Yaskawa INFORM job: DEMO_ROOF_UPPER_0625_3PAINT_58.JBI

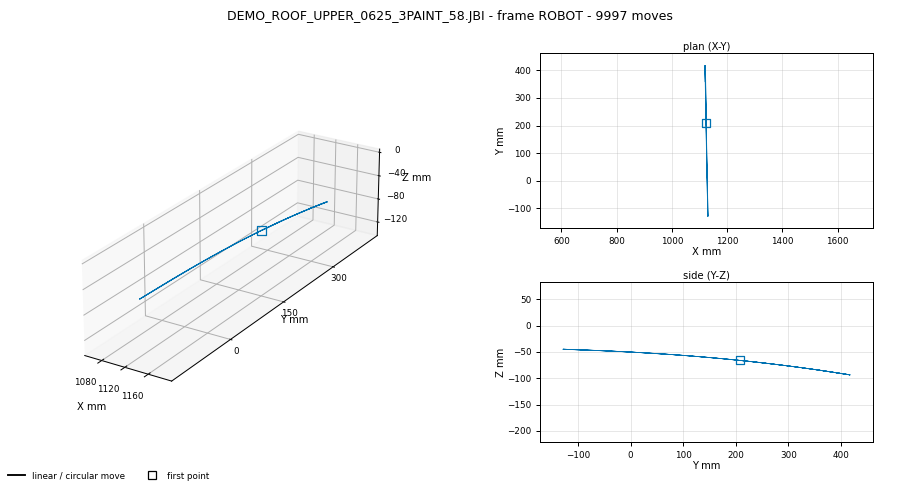
[picture p0: tool path of DEMO_ROOF_UPPER_0625_3PAINT_58.JBI in frame ROBOT, 9997 of 9997 moves have a stored position in this frame; points joined in program order, loops and branches not executed]
/JOB
//NAME DEMO_ROOF_UPPER_0625_3PAINT58
//POS
///NPOS 9997,0,0,0,0,0
///TOOL 0
///USER 0
///POSTYPE ROBOT
///RECTAN
///RCONF 1,0,0,0,0,0,0,0,0,0,0,0,0,0,0,0,0,0,0,0,0,0,0,0
C00000=1124.539,208.417,-65.917,-178.958,9.435,149.569
C00001=1124.534,208.666,-65.943,-178.955,9.438,149.569
C00002=1124.530,208.915,-65.969,-178.953,9.440,149.568
C00003=1124.525,209.163,-65.994,-178.950,9.443,149.569
C00004=1124.521,209.412,-66.020,-178.948,9.447,149.569
C00005=1124.516,209.661,-66.045,-178.945,9.449,149.568
C00006=1124.512,209.910,-66.070,-178.943,9.452,149.569
C00007=1124.507,210.158,-66.096,-178.941,9.454,149.569
C00008=1124.503,210.407,-66.122,-178.938,9.457,149.569
C00009=1124.498,210.655,-66.147,-178.937,9.459,149.569
C00010=1124.493,210.904,-66.174,-178.934,9.462,149.569
C00011=1124.489,211.153,-66.199,-178.932,9.465,149.569
C00012=1124.484,211.401,-66.225,-178.930,9.468,149.569
C00013=1124.480,211.650,-66.250,-178.928,9.470,149.569
C00014=1124.477,211.864,-66.272,-178.926,9.473,149.569
C00015=1124.472,212.078,-66.295,-178.924,9.475,149.569
C00016=1124.469,212.292,-66.316,-178.922,9.477,149.569
C00017=1124.465,212.505,-66.339,-178.920,9.480,149.569
C00018=1124.461,212.719,-66.360,-178.919,9.482,149.569
C00019=1124.457,212.933,-66.383,-178.917,9.485,149.569
C00020=1124.454,213.147,-66.405,-178.915,9.487,149.569
C00021=1124.450,213.361,-66.428,-178.914,9.489,149.570
C00022=1124.445,213.609,-66.453,-178.912,9.492,149.570
C00023=1124.441,213.858,-66.479,-178.910,9.494,149.570
C00024=1124.437,214.107,-66.505,-178.908,9.497,149.570
C00025=1124.433,214.356,-66.531,-178.906,9.500,149.570
C00026=1124.428,214.604,-66.556,-178.904,9.503,149.570
C00027=1124.423,214.853,-66.582,-178.902,9.505,149.570
C00028=1124.419,215.102,-66.608,-178.900,9.509,149.571
C00029=1124.414,215.351,-66.634,-178.898,9.511,149.571
C00030=1124.410,215.598,-66.660,-178.896,9.514,149.571
C00031=1124.406,215.847,-66.686,-178.894,9.517,149.571
C00032=1124.401,216.096,-66.711,-178.892,9.520,149.571
C00033=1124.396,216.345,-66.738,-178.890,9.522,149.571
C00034=1124.392,216.594,-66.763,-178.888,9.526,149.571
C00035=1124.387,216.842,-66.789,-178.885,9.529,149.571
C00036=1124.383,217.090,-66.815,-178.883,9.531,149.571
C00037=1124.379,217.339,-66.841,-178.881,9.535,149.572
C00038=1124.374,217.588,-66.867,-178.879,9.538,149.572
C00039=1124.370,217.837,-66.893,-178.877,9.540,149.572
C00040=1124.366,218.085,-66.920,-178.874,9.543,149.572
C00041=1124.361,218.333,-66.945,-178.872,9.547,149.572
C00042=1124.356,218.582,-66.971,-178.870,9.550,149.572
C00043=1124.352,218.830,-66.998,-178.868,9.552,149.572
C00044=1124.348,219.079,-67.024,-178.865,9.555,149.572
C00045=1124.344,219.328,-67.049,-178.863,9.559,149.573
C00046=1124.339,219.576,-67.076,-178.861,9.562,149.573
C00047=1124.335,219.825,-67.102,-178.858,9.565,149.573
C00048=1124.330,220.073,-67.128,-178.856,9.568,149.573
C00049=1124.326,220.322,-67.155,-178.853,9.571,149.573
C00050=1124.321,220.570,-67.180,-178.850,9.574,149.573
C00051=1124.317,220.819,-67.206,-178.848,9.577,149.573
C00052=1124.313,221.068,-67.233,-178.845,9.580,149.573
C00053=1124.308,221.317,-67.259,-178.843,9.584,149.573
C00054=1124.304,221.565,-67.285,-178.840,9.587,149.573
C00055=1124.299,221.814,-67.312,-178.838,9.590,149.573
C00056=1124.296,222.062,-67.338,-178.835,9.593,149.573
C00057=1124.291,222.311,-67.365,-178.832,9.597,149.573
C00058=1124.286,222.559,-67.391,-178.830,9.600,149.573
C00059=1124.282,222.807,-67.416,-178.827,9.603,149.573
C00060=1124.277,223.056,-67.443,-178.825,9.606,149.573
C00061=1124.273,223.305,-67.469,-178.822,9.609,149.573
C00062=1124.268,223.553,-67.496,-178.818,9.613,149.573
C00063=1124.264,223.802,-67.522,-178.816,9.616,149.574
C00064=1124.259,224.051,-67.549,-178.813,9.619,149.574
C00065=1124.255,224.299,-67.575,-178.810,9.623,149.574
C00066=1124.251,224.548,-67.602,-178.807,9.626,149.574
C00067=1124.247,224.796,-67.628,-178.805,9.629,149.574
C00068=1124.242,225.045,-67.655,-178.801,9.632,149.573
C00069=1124.238,225.293,-67.681,-178.799,9.635,149.574
C00070=1124.234,225.507,-67.704,-178.796,9.638,149.574
C00071=1124.230,225.721,-67.727,-178.793,9.641,149.573
C00072=1124.226,225.935,-67.750,-178.791,9.644,149.574
C00073=1124.222,226.149,-67.773,-178.788,9.647,149.573
C00074=1124.219,226.362,-67.795,-178.786,9.649,149.573
C00075=1124.215,226.576,-67.818,-178.783,9.652,149.573
C00076=1124.212,226.789,-67.842,-178.780,9.655,149.573
C00077=1124.208,227.003,-67.864,-178.777,9.658,149.573
C00078=1124.203,227.252,-67.891,-178.774,9.662,149.573
C00079=1124.199,227.500,-67.917,-178.771,9.665,149.573
C00080=1124.194,227.749,-67.944,-178.768,9.668,149.573
C00081=1124.189,227.997,-67.971,-178.765,9.672,149.573
C00082=1124.186,228.246,-67.998,-178.762,9.675,149.573
C00083=1124.181,228.494,-68.025,-178.758,9.678,149.573
C00084=1124.177,228.743,-68.051,-178.754,9.682,149.573
C00085=1124.173,228.992,-68.078,-178.751,9.684,149.573
C00086=1124.168,229.241,-68.105,-178.748,9.688,149.573
C00087=1124.164,229.489,-68.131,-178.744,9.692,149.572
C00088=1124.159,229.737,-68.159,-178.741,9.695,149.572
C00089=1124.155,229.986,-68.186,-178.738,9.698,149.572
C00090=1124.150,230.234,-68.213,-178.734,9.701,149.572
C00091=1124.146,230.482,-68.239,-178.731,9.705,149.572
C00092=1124.141,230.731,-68.266,-178.727,9.708,149.572
C00093=1124.137,230.979,-68.293,-178.724,9.711,149.572
C00094=1124.133,231.228,-68.320,-178.721,9.715,149.572
C00095=1124.129,231.477,-68.347,-178.718,9.717,149.572
C00096=1124.124,231.725,-68.374,-178.714,9.721,149.571
C00097=1124.120,231.974,-68.401,-178.711,9.723,149.571
C00098=1124.115,232.222,-68.428,-178.707,9.727,149.571
C00099=1124.111,232.470,-68.455,-178.704,9.730,149.571
C00100=1124.107,232.720,-68.482,-178.701,9.732,149.571
C00101=1124.103,232.967,-68.510,-178.698,9.736,149.571
C00102=1124.098,233.216,-68.537,-178.695,9.739,149.570
C00103=1124.093,233.464,-68.564,-178.692,9.741,149.570
C00104=1124.089,233.713,-68.591,-178.689,9.744,149.570
C00105=1124.085,233.962,-68.618,-178.686,9.747,149.570
C00106=1124.081,234.210,-68.645,-178.682,9.750,149.570
C00107=1124.076,234.458,-68.673,-178.679,9.753,149.570
C00108=1124.072,234.707,-68.700,-178.676,9.756,149.570
C00109=1124.068,234.956,-68.727,-178.673,9.759,149.570
C00110=1124.063,235.204,-68.754,-178.670,9.761,149.569
C00111=1124.059,235.452,-68.782,-178.668,9.764,149.570
C00112=1124.054,235.701,-68.809,-178.665,9.767,149.569
C00113=1124.051,235.950,-68.836,-178.662,9.770,149.569
C00114=1124.046,236.198,-68.864,-178.660,9.772,149.569
C00115=1124.042,236.446,-68.891,-178.657,9.775,149.569
C00116=1124.037,236.695,-68.918,-178.654,9.777,149.569
C00117=1124.033,236.943,-68.946,-178.651,9.780,149.569
C00118=1124.028,237.192,-68.973,-178.648,9.783,149.569
C00119=1124.024,237.440,-69.000,-178.646,9.785,149.569
C00120=1124.019,237.688,-69.028,-178.643,9.788,149.569
C00121=1124.015,237.937,-69.055,-178.640,9.791,149.568
C00122=1124.011,238.185,-69.083,-178.638,9.793,149.568
C00123=1124.006,238.434,-69.110,-178.635,9.796,149.568
C00124=1124.003,238.682,-69.138,-178.632,9.799,149.568
C00125=1123.998,238.931,-69.165,-178.630,9.801,149.568
C00126=1123.994,239.145,-69.190,-178.628,9.803,149.568
C00127=1123.990,239.358,-69.213,-178.626,9.805,149.568
C00128=1123.986,239.571,-69.236,-178.624,9.807,149.568
C00129=1123.983,239.785,-69.260,-178.622,9.809,149.568
C00130=1123.979,239.998,-69.284,-178.620,9.811,149.568
C00131=1123.976,240.212,-69.308,-178.617,9.813,149.568
C00132=1123.972,240.426,-69.331,-178.616,9.816,149.568
C00133=1123.968,240.640,-69.355,-178.613,9.818,149.568
C00134=1123.963,240.888,-69.383,-178.611,9.820,149.568
C00135=1123.959,241.137,-69.411,-178.609,9.822,149.568
C00136=1123.955,241.385,-69.438,-178.606,9.825,149.568
C00137=1123.951,241.633,-69.466,-178.604,9.827,149.568
C00138=1123.947,241.882,-69.494,-178.602,9.829,149.568
C00139=1123.942,242.130,-69.521,-178.600,9.832,149.568
C00140=1123.937,242.379,-69.549,-178.597,9.835,149.568
C00141=1123.933,242.627,-69.577,-178.596,9.837,149.568
C00142=1123.929,242.875,-69.605,-178.594,9.839,149.568
C00143=1123.925,243.124,-69.632,-178.592,9.842,149.568
C00144=1123.920,243.372,-69.660,-178.590,9.844,149.568
C00145=1123.917,243.621,-69.688,-178.588,9.846,149.568
C00146=1123.912,243.869,-69.715,-178.586,9.848,149.568
C00147=1123.907,244.117,-69.744,-178.584,9.851,149.568
C00148=1123.903,244.366,-69.772,-178.582,9.853,149.568
C00149=1123.898,244.614,-69.799,-178.580,9.855,149.568
C00150=1123.895,244.863,-69.827,-178.578,9.858,149.568
C00151=1123.890,245.111,-69.855,-178.577,9.860,149.568
C00152=1123.886,245.360,-69.884,-178.575,9.863,149.568
C00153=1123.881,245.608,-69.911,-178.573,9.865,149.568
C00154=1123.877,245.856,-69.938,-178.572,9.866,149.568
C00155=1123.873,246.105,-69.967,-178.570,9.869,149.569
C00156=1123.869,246.353,-69.994,-178.568,9.871,149.569
C00157=1123.864,246.602,-70.022,-178.566,9.874,149.569
C00158=1123.860,246.850,-70.050,-178.565,9.876,149.569
C00159=1123.856,247.099,-70.078,-178.563,9.878,149.569
C00160=1123.851,247.346,-70.106,-178.562,9.881,149.569
C00161=1123.847,247.595,-70.135,-178.557,9.885,149.569
C00162=1123.842,247.844,-70.162,-178.552,9.889,149.569
C00163=1123.838,248.092,-70.190,-178.545,9.894,149.568
C00164=1123.833,248.341,-70.218,-178.540,9.899,149.568
C00165=1123.829,248.588,-70.246,-178.534,9.903,149.568
C00166=1123.825,248.837,-70.274,-178.529,9.908,149.567
C00167=1123.821,249.086,-70.303,-178.524,9.911,149.567
C00168=1123.817,249.334,-70.331,-178.519,9.915,149.566
C00169=1123.813,249.582,-70.359,-178.513,9.920,149.566
C00170=1123.808,249.831,-70.387,-178.509,9.923,149.566
C00171=1123.804,250.079,-70.415,-178.505,9.927,149.565
C00172=1123.799,250.327,-70.444,-178.500,9.931,149.565
C00173=1123.795,250.576,-70.472,-178.496,9.933,149.565
C00174=1123.790,250.824,-70.500,-178.492,9.937,149.564
C00175=1123.787,251.072,-70.529,-178.489,9.939,149.564
C00176=1123.783,251.321,-70.557,-178.485,9.943,149.564
C00177=1123.778,251.569,-70.586,-178.482,9.945,149.564
C00178=1123.774,251.817,-70.614,-178.478,9.948,149.563
C00179=1123.769,252.066,-70.642,-178.475,9.950,149.563
C00180=1123.765,252.313,-70.671,-178.472,9.953,149.563
C00181=1123.761,252.562,-70.700,-178.469,9.956,149.563
C00182=1123.756,252.776,-70.724,-178.467,9.958,149.563
C00183=1123.754,252.989,-70.748,-178.465,9.959,149.563
C00184=1123.750,253.203,-70.773,-178.463,9.961,149.563
C00185=1123.746,253.417,-70.797,-178.462,9.962,149.562
C00186=1123.742,253.629,-70.822,-178.460,9.965,149.563
C00187=1123.739,253.843,-70.846,-178.458,9.966,149.562
C00188=1123.735,254.057,-70.871,-178.457,9.967,149.562
C00189=1123.731,254.271,-70.896,-178.456,9.969,149.562
C00190=1123.727,254.518,-70.924,-178.455,9.970,149.563
C00191=1123.723,254.767,-70.953,-178.454,9.972,149.563
C00192=1123.719,255.016,-70.981,-178.453,9.973,149.563
C00193=1123.714,255.263,-71.010,-178.453,9.974,149.563
C00194=1123.710,255.512,-71.039,-178.453,9.975,149.563
C00195=1123.705,255.760,-71.067,-178.452,9.977,149.563
C00196=1123.701,256.008,-71.096,-178.451,9.978,149.564
C00197=1123.697,256.257,-71.124,-178.449,9.981,149.564
C00198=1123.692,256.505,-71.153,-178.446,9.984,149.563
C00199=1123.689,256.753,-71.182,-178.443,9.987,149.564
C00200=1123.684,257.002,-71.210,-178.440,9.990,149.563
C00201=1123.680,257.251,-71.239,-178.437,9.993,149.563
C00202=1123.676,257.498,-71.268,-178.434,9.995,149.563
C00203=1123.671,257.747,-71.296,-178.431,9.998,149.563
C00204=1123.667,257.995,-71.326,-178.428,10.001,149.563
C00205=1123.663,258.243,-71.353,-178.425,10.004,149.563
C00206=1123.658,258.492,-71.382,-178.422,10.006,149.563
C00207=1123.654,258.740,-71.412,-178.420,10.009,149.563
C00208=1123.650,258.988,-71.439,-178.416,10.013,149.563
C00209=1123.646,259.236,-71.469,-178.413,10.015,149.562
C00210=1123.641,259.485,-71.498,-178.410,10.018,149.562
C00211=1123.638,259.733,-71.526,-178.407,10.021,149.562
C00212=1123.633,259.981,-71.555,-178.404,10.024,149.562
C00213=1123.628,260.229,-71.584,-178.401,10.027,149.562
C00214=1123.624,260.478,-71.614,-178.398,10.030,149.562
C00215=1123.620,260.726,-71.642,-178.394,10.034,149.562
C00216=1123.616,260.975,-71.671,-178.391,10.036,149.562
C00217=1123.611,261.223,-71.700,-178.388,10.039,149.561
C00218=1123.607,261.471,-71.729,-178.384,10.042,149.561
C00219=1123.603,261.719,-71.759,-178.381,10.045,149.561
C00220=1123.599,261.968,-71.787,-178.377,10.048,149.561
C00221=1123.595,262.216,-71.816,-178.374,10.051,149.561
C00222=1123.590,262.464,-71.845,-178.370,10.054,149.561
C00223=1123.586,262.713,-71.874,-178.367,10.057,149.560
C00224=1123.581,262.961,-71.904,-178.363,10.060,149.560
C00225=1123.577,263.209,-71.933,-178.360,10.063,149.560
C00226=1123.574,263.457,-71.962,-178.357,10.066,149.560
C00227=1123.569,263.705,-71.990,-178.354,10.069,149.560
C00228=1123.565,263.954,-72.020,-178.350,10.072,149.559
C00229=1123.560,264.202,-72.049,-178.346,10.075,149.559
C00230=1123.556,264.450,-72.079,-178.343,10.078,149.559
C00231=1123.552,264.698,-72.108,-178.340,10.081,149.559
C00232=1123.548,264.947,-72.137,-178.337,10.083,149.559
C00233=1123.543,265.196,-72.166,-178.334,10.085,149.559
C00234=1123.539,265.443,-72.195,-178.332,10.087,149.559
C00235=1123.534,265.691,-72.225,-178.329,10.090,149.558
C00236=1123.530,265.940,-72.254,-178.327,10.092,149.558
C00237=1123.526,266.188,-72.284,-178.324,10.095,149.558
C00238=1123.522,266.401,-72.309,-178.322,10.097,149.558
C00239=1123.519,266.615,-72.334,-178.319,10.099,149.558
C00240=1123.515,266.828,-72.359,-178.317,10.101,149.558
C00241=1123.512,267.042,-72.384,-178.315,10.103,149.558
C00242=1123.508,267.255,-72.410,-178.313,10.105,149.558
C00243=1123.505,267.468,-72.435,-178.311,10.107,149.558
C00244=1123.501,267.682,-72.460,-178.308,10.109,149.558
C00245=1123.498,267.895,-72.486,-178.306,10.111,149.558
C00246=1123.494,268.143,-72.515,-178.303,10.114,149.558
C00247=1123.489,268.390,-72.544,-178.300,10.117,149.557
C00248=1123.485,268.639,-72.574,-178.298,10.119,149.557
C00249=1123.480,268.887,-72.604,-178.295,10.122,149.557
C00250=1123.476,269.136,-72.633,-178.292,10.124,149.557
C00251=1123.471,269.384,-72.663,-178.290,10.126,149.557
C00252=1123.467,269.632,-72.692,-178.287,10.129,149.557
C00253=1123.463,269.880,-72.722,-178.284,10.132,149.557
C00254=1123.459,270.129,-72.751,-178.281,10.135,149.557
C00255=1123.455,270.377,-72.781,-178.279,10.137,149.557
C00256=1123.450,270.625,-72.810,-178.276,10.139,149.556
C00257=1123.447,270.873,-72.840,-178.273,10.142,149.556
C00258=1123.442,271.121,-72.870,-178.270,10.145,149.556
C00259=1123.438,271.369,-72.899,-178.268,10.147,149.556
C00260=1123.433,271.618,-72.929,-178.265,10.150,149.556
C00261=1123.429,271.866,-72.959,-178.262,10.152,149.556
C00262=1123.425,272.114,-72.988,-178.259,10.155,149.556
C00263=1123.421,272.362,-73.018,-178.256,10.158,149.556
C00264=1123.417,272.610,-73.048,-178.253,10.160,149.555
C00265=1123.413,272.859,-73.077,-178.250,10.163,149.555
C00266=1123.408,273.107,-73.108,-178.247,10.166,149.555
C00267=1123.404,273.355,-73.137,-178.244,10.169,149.555
C00268=1123.400,273.603,-73.167,-178.241,10.171,149.555
C00269=1123.396,273.851,-73.196,-178.239,10.173,149.555
C00270=1123.392,274.100,-73.227,-178.236,10.176,149.555
C00271=1123.387,274.348,-73.257,-178.232,10.179,149.555
C00272=1123.383,274.597,-73.286,-178.229,10.181,149.554
C00273=1123.379,274.844,-73.316,-178.226,10.184,149.554
C00274=1123.375,275.093,-73.346,-178.223,10.187,149.554
C00275=1123.370,275.340,-73.377,-178.221,10.190,149.554
C00276=1123.366,275.589,-73.406,-178.217,10.192,149.554
C00277=1123.362,275.837,-73.436,-178.214,10.196,149.554
C00278=1123.358,276.085,-73.466,-178.211,10.198,149.554
C00279=1123.353,276.333,-73.496,-178.208,10.201,149.554
C00280=1123.350,276.582,-73.526,-178.204,10.203,149.553
C00281=1123.346,276.830,-73.556,-178.201,10.206,149.553
C00282=1123.341,277.078,-73.587,-178.199,10.209,149.553
C00283=1123.337,277.326,-73.616,-178.195,10.211,149.553
C00284=1123.333,277.574,-73.646,-178.192,10.214,149.553
C00285=1123.328,277.822,-73.676,-178.189,10.217,149.552
C00286=1123.324,278.070,-73.706,-178.185,10.220,149.552
C00287=1123.320,278.319,-73.738,-178.182,10.223,149.552
C00288=1123.316,278.567,-73.767,-178.179,10.225,149.552
C00289=1123.312,278.815,-73.797,-178.176,10.228,149.552
C00290=1123.307,279.063,-73.827,-178.173,10.230,149.552
C00291=1123.304,279.311,-73.857,-178.169,10.234,149.552
C00292=1123.299,279.559,-73.888,-178.166,10.236,149.551
C00293=1123.295,279.808,-73.918,-178.163,10.239,149.551
C00294=1123.291,280.021,-73.944,-178.160,10.242,149.551
C00295=1123.288,280.234,-73.970,-178.157,10.244,149.551
C00296=1123.285,280.447,-73.996,-178.154,10.246,149.551
C00297=1123.281,280.660,-74.022,-178.151,10.249,149.550
C00298=1123.277,280.873,-74.048,-178.149,10.251,149.550
C00299=1123.274,281.087,-74.075,-178.145,10.253,149.550
C00300=1123.270,281.300,-74.101,-178.142,10.256,149.550
C00301=1123.266,281.513,-74.126,-178.140,10.258,149.550
C00302=1123.262,281.761,-74.157,-178.137,10.260,149.549
C00303=1123.258,282.009,-74.187,-178.134,10.263,149.549
C00304=1123.254,282.258,-74.219,-178.130,10.265,149.549
C00305=1123.250,282.506,-74.248,-178.128,10.268,149.549
C00306=1123.245,282.754,-74.279,-178.124,10.271,149.549
C00307=1123.241,283.001,-74.309,-178.121,10.273,149.549
C00308=1123.237,283.250,-74.340,-178.118,10.276,149.548
C00309=1123.233,283.498,-74.370,-178.115,10.279,149.548
C00310=1123.229,283.746,-74.401,-178.113,10.281,149.548
C00311=1123.224,283.994,-74.432,-178.109,10.283,149.548
C00312=1123.221,284.242,-74.462,-178.106,10.286,149.548
C00313=1123.216,284.490,-74.493,-178.103,10.288,149.547
C00314=1123.212,284.738,-74.523,-178.100,10.291,149.547
C00315=1123.208,284.987,-74.554,-178.097,10.294,149.547
C00316=1123.203,285.235,-74.584,-178.094,10.296,149.547
C00317=1123.199,285.482,-74.615,-178.091,10.299,149.547
C00318=1123.195,285.731,-74.646,-178.088,10.301,149.547
C00319=1123.191,285.979,-74.676,-178.085,10.303,149.546
C00320=1123.187,286.227,-74.707,-178.082,10.306,149.546
C00321=1123.183,286.475,-74.738,-178.079,10.308,149.546
C00322=1123.179,286.723,-74.769,-178.076,10.311,149.546
C00323=1123.175,286.970,-74.799,-178.073,10.314,149.546
C00324=1123.171,287.219,-74.831,-178.070,10.316,149.546
C00325=1123.166,287.467,-74.861,-178.066,10.319,149.545
C00326=1123.162,287.715,-74.892,-178.063,10.322,149.545
C00327=1123.158,287.963,-74.923,-178.060,10.324,149.545
C00328=1123.154,288.211,-74.953,-178.057,10.327,149.545
C00329=1123.149,288.459,-74.984,-178.054,10.328,149.545
C00330=1123.145,288.707,-75.016,-178.052,10.331,149.545
C00331=1123.141,288.955,-75.046,-178.049,10.334,149.544
C00332=1123.137,289.204,-75.077,-178.045,10.336,149.544
C00333=1123.133,289.451,-75.108,-178.042,10.339,149.544
C00334=1123.128,289.699,-75.139,-178.039,10.342,149.544
C00335=1123.124,289.947,-75.171,-178.036,10.344,149.544
C00336=1123.121,290.195,-75.201,-178.033,10.347,149.543
C00337=1123.117,290.444,-75.232,-178.030,10.349,149.543
C00338=1123.112,290.692,-75.263,-178.026,10.352,149.543
C00339=1123.108,290.940,-75.295,-178.024,10.354,149.543
C00340=1123.104,291.188,-75.325,-178.021,10.356,149.543
C00341=1123.100,291.436,-75.356,-178.018,10.359,149.543
C00342=1123.096,291.683,-75.387,-178.015,10.362,149.543
C00343=1123.091,291.931,-75.418,-178.012,10.364,149.542
C00344=1123.087,292.180,-75.449,-178.009,10.367,149.542
C00345=1123.083,292.427,-75.481,-178.005,10.369,149.542
C00346=1123.079,292.676,-75.512,-178.002,10.372,149.542
C00347=1123.075,292.923,-75.543,-177.999,10.375,149.542
C00348=1123.071,293.172,-75.574,-177.996,10.377,149.541
C00349=1123.067,293.419,-75.606,-177.993,10.380,149.541
C00350=1123.064,293.633,-75.632,-177.990,10.382,149.541
C00351=1123.060,293.846,-75.659,-177.988,10.384,149.541
C00352=1123.057,294.059,-75.686,-177.985,10.386,149.541
C00353=1123.053,294.272,-75.713,-177.983,10.388,149.541
C00354=1123.049,294.485,-75.740,-177.980,10.390,149.540
C00355=1123.046,294.699,-75.767,-177.977,10.393,149.540
C00356=1123.042,294.911,-75.794,-177.975,10.395,149.540
C00357=1123.039,295.125,-75.821,-177.972,10.397,149.540
C00358=1123.034,295.372,-75.852,-177.969,10.399,149.540
C00359=1123.030,295.621,-75.883,-177.966,10.402,149.540
C00360=1123.026,295.868,-75.915,-177.963,10.405,149.539
C00361=1123.022,296.117,-75.946,-177.960,10.407,149.539
C00362=1123.018,296.364,-75.978,-177.957,10.410,149.539
C00363=1123.014,296.613,-76.009,-177.953,10.412,149.539
C00364=1123.009,296.860,-76.040,-177.951,10.415,149.539
C00365=1123.006,297.108,-76.072,-177.947,10.417,149.539
C00366=1123.002,297.357,-76.103,-177.944,10.420,149.538
C00367=1122.997,297.604,-76.135,-177.942,10.422,149.538
C00368=1122.994,297.852,-76.166,-177.939,10.425,149.538
C00369=1122.989,298.100,-76.197,-177.935,10.427,149.538
C00370=1122.985,298.348,-76.229,-177.932,10.430,149.538
C00371=1122.981,298.596,-76.261,-177.929,10.432,149.537
C00372=1122.977,298.844,-76.292,-177.926,10.435,149.537
C00373=1122.973,299.093,-76.324,-177.923,10.437,149.537
C00374=1122.968,299.340,-76.356,-177.920,10.440,149.537
C00375=1122.965,299.588,-76.387,-177.917,10.443,149.537
C00376=1122.961,299.836,-76.419,-177.914,10.445,149.537
C00377=1122.957,300.083,-76.451,-177.910,10.448,149.536
C00378=1122.952,300.332,-76.482,-177.908,10.450,149.536
C00379=1122.948,300.580,-76.514,-177.905,10.452,149.536
C00380=1122.944,300.828,-76.546,-177.902,10.455,149.536
C00381=1122.940,301.076,-76.578,-177.898,10.457,149.536
C00382=1122.936,301.323,-76.609,-177.895,10.460,149.536
C00383=1122.932,301.571,-76.641,-177.892,10.463,149.535
C00384=1122.928,301.820,-76.673,-177.889,10.465,149.535
C00385=1122.923,302.067,-76.705,-177.886,10.468,149.535
C00386=1122.919,302.316,-76.736,-177.883,10.471,149.535
C00387=1122.915,302.564,-76.768,-177.880,10.473,149.535
C00388=1122.911,302.811,-76.800,-177.877,10.476,149.535
C00389=1122.907,303.059,-76.832,-177.873,10.478,149.534
C00390=1122.903,303.307,-76.864,-177.871,10.480,149.534
C00391=1122.899,303.556,-76.896,-177.868,10.483,149.534
C00392=1122.894,303.803,-76.928,-177.864,10.485,149.534
C00393=1122.891,304.051,-76.959,-177.861,10.488,149.534
C00394=1122.886,304.299,-76.992,-177.858,10.490,149.533
C00395=1122.882,304.547,-77.023,-177.855,10.493,149.533
C00396=1122.878,304.794,-77.056,-177.852,10.495,149.533
C00397=1122.874,305.042,-77.088,-177.849,10.498,149.533
C00398=1122.870,305.290,-77.120,-177.846,10.501,149.533
C00399=1122.866,305.538,-77.152,-177.843,10.503,149.533
C00400=1122.862,305.786,-77.184,-177.839,10.506,149.532
C00401=1122.858,306.034,-77.216,-177.836,10.509,149.532
C00402=1122.853,306.283,-77.248,-177.834,10.510,149.532
C00403=1122.849,306.530,-77.280,-177.831,10.513,149.532
C00404=1122.846,306.777,-77.312,-177.827,10.516,149.532
C00405=1122.841,307.026,-77.345,-177.824,10.518,149.531
C00406=1122.838,307.238,-77.372,-177.821,10.521,149.531
C00407=1122.834,307.451,-77.400,-177.819,10.523,149.531
C00408=1122.831,307.665,-77.428,-177.816,10.524,149.531
C00409=1122.827,307.877,-77.455,-177.813,10.527,149.531
C00410=1122.824,308.091,-77.483,-177.811,10.529,149.531
C00411=1122.820,308.303,-77.511,-177.808,10.531,149.530
C00412=1122.817,308.516,-77.539,-177.805,10.534,149.530
C00413=1122.814,308.729,-77.566,-177.803,10.536,149.530
C00414=1122.809,308.977,-77.599,-177.800,10.538,149.530
C00415=1122.805,309.225,-77.630,-177.797,10.541,149.530
C00416=1122.801,309.472,-77.663,-177.793,10.543,149.530
C00417=1122.797,309.721,-77.695,-177.790,10.546,149.529
C00418=1122.793,309.968,-77.728,-177.787,10.548,149.529
C00419=1122.789,310.216,-77.760,-177.784,10.551,149.529
C00420=1122.785,310.465,-77.793,-177.781,10.554,149.529
C00421=1122.781,310.711,-77.825,-177.778,10.556,149.529
C00422=1122.776,310.960,-77.857,-177.775,10.558,149.529
C00423=1122.773,311.207,-77.890,-177.772,10.560,149.528
C00424=1122.768,311.455,-77.922,-177.769,10.563,149.528
C00425=1122.764,311.703,-77.955,-177.766,10.566,149.528
C00426=1122.761,311.951,-77.987,-177.762,10.568,149.528
C00427=1122.756,312.200,-78.020,-177.759,10.571,149.528
C00428=1122.753,312.447,-78.052,-177.756,10.573,149.527
C00429=1122.749,312.695,-78.085,-177.753,10.576,149.527
C00430=1122.744,312.943,-78.118,-177.750,10.579,149.527
C00431=1122.740,313.190,-78.150,-177.746,10.581,149.527
C00432=1122.736,313.438,-78.182,-177.744,10.584,149.527
C00433=1122.732,313.686,-78.215,-177.740,10.586,149.526
C00434=1122.728,313.934,-78.247,-177.737,10.589,149.526
C00435=1122.724,314.182,-78.281,-177.735,10.591,149.526
C00436=1122.720,314.429,-78.313,-177.731,10.593,149.526
C00437=1122.716,314.677,-78.346,-177.728,10.596,149.526
C00438=1122.712,314.925,-78.379,-177.725,10.598,149.526
C00439=1122.708,315.173,-78.411,-177.722,10.601,149.525
C00440=1122.704,315.421,-78.444,-177.719,10.603,149.525
C00441=1122.700,315.669,-78.477,-177.715,10.606,149.525
C00442=1122.696,315.916,-78.510,-177.712,10.609,149.525
C00443=1122.692,316.164,-78.542,-177.709,10.611,149.525
C00444=1122.688,316.412,-78.575,-177.706,10.614,149.525
C00445=1122.684,316.660,-78.608,-177.703,10.616,149.524
C00446=1122.679,316.908,-78.641,-177.700,10.619,149.524
C00447=1122.676,317.156,-78.673,-177.697,10.622,149.524
C00448=1122.672,317.403,-78.706,-177.693,10.624,149.524
C00449=1122.668,317.651,-78.740,-177.691,10.626,149.524
C00450=1122.663,317.899,-78.773,-177.688,10.628,149.523
C00451=1122.660,318.146,-78.805,-177.684,10.631,149.523
C00452=1122.656,318.394,-78.838,-177.681,10.634,149.523
C00453=1122.651,318.642,-78.871,-177.678,10.636,149.523
C00454=1122.647,318.890,-78.904,-177.675,10.639,149.523
C00455=1122.643,319.138,-78.937,-177.672,10.641,149.522
C00456=1122.639,319.386,-78.970,-177.669,10.644,149.522
C00457=1122.636,319.633,-79.003,-177.666,10.647,149.522
C00458=1122.632,319.881,-79.036,-177.662,10.649,149.522
C00459=1122.628,320.129,-79.070,-177.659,10.651,149.522
C00460=1122.624,320.377,-79.103,-177.656,10.654,149.522
C00461=1122.620,320.625,-79.136,-177.653,10.657,149.521
C00462=1122.617,320.837,-79.164,-177.650,10.659,149.521
C00463=1122.613,321.049,-79.193,-177.648,10.660,149.521
C00464=1122.609,321.263,-79.221,-177.645,10.663,149.521
C00465=1122.606,321.475,-79.249,-177.642,10.665,149.521
C00466=1122.603,321.688,-79.278,-177.640,10.667,149.521
C00467=1122.599,321.901,-79.307,-177.637,10.670,149.520
C00468=1122.596,322.114,-79.335,-177.634,10.671,149.520
C00469=1122.592,322.327,-79.363,-177.631,10.674,149.520
C00470=1122.589,322.574,-79.397,-177.628,10.676,149.520
C00471=1122.584,322.822,-79.430,-177.625,10.678,149.520
C00472=1122.580,323.070,-79.464,-177.622,10.681,149.520
C00473=1122.576,323.318,-79.497,-177.619,10.683,149.519
C00474=1122.571,323.621,-79.538,-177.615,10.687,149.519
C00475=1122.567,323.924,-79.578,-177.611,10.690,149.519
C00476=1122.561,324.227,-79.619,-177.607,10.693,149.519
C00477=1122.557,324.530,-79.660,-177.603,10.696,149.518
C00478=1122.553,324.777,-79.693,-177.600,10.699,149.518
C00479=1122.549,325.025,-79.726,-177.598,10.701,149.518
C00480=1122.545,325.273,-79.760,-177.594,10.703,149.518
C00481=1122.541,325.521,-79.793,-177.591,10.706,149.518
C00482=1122.536,325.769,-79.827,-177.588,10.708,149.518
C00483=1122.533,326.016,-79.861,-177.585,10.711,149.517
C00484=1122.528,326.264,-79.894,-177.581,10.713,149.517
C00485=1122.525,326.512,-79.928,-177.578,10.716,149.517
C00486=1122.521,326.759,-79.962,-177.575,10.718,149.517
C00487=1122.517,327.007,-79.995,-177.572,10.721,149.516
C00488=1122.513,327.255,-80.028,-177.568,10.723,149.516
C00489=1122.509,327.502,-80.062,-177.566,10.726,149.516
C00490=1122.505,327.750,-80.096,-177.562,10.729,149.516
C00491=1122.501,327.998,-80.129,-177.559,10.731,149.516
C00492=1122.497,328.245,-80.163,-177.556,10.734,149.516
C00493=1122.493,328.493,-80.196,-177.553,10.735,149.515
C00494=1122.489,328.741,-80.230,-177.550,10.738,149.515
C00495=1122.485,328.989,-80.263,-177.547,10.741,149.515
C00496=1122.481,329.236,-80.298,-177.544,10.743,149.515
C00497=1122.476,329.484,-80.331,-177.540,10.746,149.515
C00498=1122.473,329.732,-80.365,-177.537,10.748,149.514
C00499=1122.469,329.979,-80.399,-177.534,10.751,149.514
C00500=1122.465,330.227,-80.433,-177.531,10.753,149.514
C00501=1122.461,330.475,-80.466,-177.528,10.756,149.514
C00502=1122.457,330.722,-80.500,-177.525,10.758,149.514
C00503=1122.453,330.970,-80.534,-177.521,10.761,149.513
C00504=1122.449,331.218,-80.568,-177.518,10.763,149.513
C00505=1122.445,331.465,-80.602,-177.515,10.766,149.513
C00506=1122.441,331.713,-80.635,-177.512,10.769,149.513
C00507=1122.437,331.960,-80.669,-177.508,10.771,149.513
C00508=1122.433,332.209,-80.703,-177.505,10.773,149.512
C00509=1122.429,332.456,-80.737,-177.503,10.775,149.512
C00510=1122.426,332.704,-80.771,-177.499,10.778,149.512
C00511=1122.421,332.952,-80.805,-177.496,10.780,149.512
C00512=1122.417,333.199,-80.839,-177.493,10.783,149.512
C00513=1122.414,333.447,-80.873,-177.490,10.786,149.512
C00514=1122.409,333.694,-80.908,-177.487,10.788,149.511
C00515=1122.405,333.942,-80.941,-177.483,10.791,149.511
C00516=1122.402,334.190,-80.975,-177.480,10.793,149.511
C00517=1122.397,334.437,-81.010,-177.477,10.796,149.511
C00518=1122.392,334.808,-81.060,-177.472,10.799,149.510
C00519=1122.386,335.177,-81.112,-177.467,10.803,149.510
C00520=1122.381,335.547,-81.163,-177.463,10.807,149.510
C00521=1122.374,335.917,-81.214,-177.458,10.810,149.510
C00522=1122.370,336.164,-81.247,-177.455,10.812,149.509
C00523=1122.366,336.412,-81.282,-177.452,10.815,149.509
C00524=1122.362,336.659,-81.316,-177.449,10.818,149.509
C00525=1122.358,336.907,-81.351,-177.445,10.820,149.509
C00526=1122.354,337.155,-81.385,-177.442,10.823,149.509
C00527=1122.350,337.403,-81.420,-177.439,10.825,149.508
C00528=1122.347,337.650,-81.454,-177.436,10.828,149.508
C00529=1122.343,337.898,-81.488,-177.432,10.830,149.508
C00530=1122.339,338.145,-81.522,-177.429,10.833,149.508
C00531=1122.334,338.392,-81.557,-177.426,10.836,149.508
C00532=1122.331,338.640,-81.591,-177.423,10.838,149.507
C00533=1122.326,338.888,-81.625,-177.420,10.840,149.507
C00534=1122.323,339.135,-81.660,-177.416,10.843,149.507
C00535=1122.319,339.383,-81.694,-177.413,10.845,149.507
C00536=1122.315,339.631,-81.729,-177.410,10.848,149.507
C00537=1122.311,339.878,-81.763,-177.407,10.850,149.506
C00538=1122.307,340.126,-81.798,-177.404,10.852,149.506
C00539=1122.303,340.373,-81.832,-177.401,10.855,149.506
C00540=1122.299,340.621,-81.866,-177.397,10.857,149.506
C00541=1122.295,340.869,-81.901,-177.394,10.860,149.506
C00542=1122.291,341.117,-81.935,-177.391,10.862,149.505
C00543=1122.287,341.363,-81.970,-177.388,10.865,149.505
C00544=1122.283,341.612,-82.005,-177.385,10.867,149.505
C00545=1122.279,341.859,-82.039,-177.381,10.870,149.505
C00546=1122.275,342.107,-82.074,-177.378,10.873,149.505
C00547=1122.271,342.354,-82.109,-177.375,10.875,149.504
C00548=1122.268,342.601,-82.143,-177.372,10.877,149.504
C00549=1122.264,342.850,-82.178,-177.368,10.880,149.504
C00550=1122.259,343.097,-82.213,-177.365,10.882,149.504
C00551=1122.256,343.344,-82.247,-177.362,10.885,149.504
C00552=1122.252,343.592,-82.282,-177.359,10.888,149.504
C00553=1122.248,343.840,-82.317,-177.356,10.889,149.503
C00554=1122.244,344.086,-82.352,-177.353,10.892,149.503
C00555=1122.240,344.334,-82.386,-177.349,10.894,149.503
C00556=1122.236,344.582,-82.421,-177.346,10.897,149.503
C00557=1122.232,344.829,-82.456,-177.343,10.899,149.503
C00558=1122.228,345.077,-82.491,-177.340,10.902,149.502
C00559=1122.224,345.324,-82.525,-177.337,10.904,149.502
C00560=1122.221,345.572,-82.560,-177.333,10.907,149.502
C00561=1122.217,345.820,-82.595,-177.330,10.909,149.502
C00562=1122.212,346.067,-82.630,-177.327,10.912,149.501
C00563=1122.208,346.315,-82.665,-177.324,10.915,149.501
C00564=1122.205,346.562,-82.701,-177.320,10.917,149.501
C00565=1122.201,346.810,-82.735,-177.317,10.919,149.501
C00566=1122.197,347.057,-82.770,-177.314,10.922,149.501
C00567=1122.193,347.305,-82.805,-177.311,10.924,149.500
C00568=1122.189,347.552,-82.840,-177.307,10.927,149.500
C00569=1122.185,347.800,-82.875,-177.304,10.929,149.500
C00570=1122.182,348.012,-82.905,-177.302,10.931,149.500
C00571=1122.178,348.224,-82.936,-177.299,10.933,149.500
C00572=1122.176,348.437,-82.966,-177.296,10.936,149.500
C00573=1122.172,348.650,-82.996,-177.293,10.937,149.499
C00574=1122.168,348.862,-83.025,-177.291,10.939,149.499
C00575=1122.165,349.075,-83.056,-177.288,10.942,149.499
C00576=1122.162,349.287,-83.086,-177.285,10.944,149.499
C00577=1122.158,349.500,-83.116,-177.282,10.946,149.499
C00578=1122.155,349.747,-83.152,-177.279,10.949,149.498
C00579=1122.151,349.995,-83.187,-177.275,10.951,149.498
C00580=1122.146,350.242,-83.222,-177.272,10.953,149.498
C00581=1122.143,350.489,-83.257,-177.268,10.957,149.498
C00582=1122.139,350.737,-83.292,-177.265,10.959,149.497
C00583=1122.136,350.985,-83.327,-177.261,10.962,149.497
C00584=1122.131,351.232,-83.363,-177.258,10.964,149.497
C00585=1122.128,351.479,-83.398,-177.255,10.967,149.497
C00586=1122.124,351.727,-83.433,-177.250,10.969,149.496
C00587=1122.120,351.975,-83.468,-177.247,10.972,149.496
C00588=1122.116,352.222,-83.504,-177.244,10.974,149.496
C00589=1122.112,352.469,-83.539,-177.240,10.977,149.496
C00590=1122.108,352.717,-83.575,-177.237,10.979,149.495
C00591=1122.104,352.964,-83.611,-177.233,10.983,149.495
C00592=1122.100,353.211,-83.646,-177.229,10.985,149.495
C00593=1122.096,353.459,-83.681,-177.226,10.987,149.495
C00594=1122.092,353.707,-83.716,-177.223,10.990,149.494
C00595=1122.089,353.954,-83.752,-177.219,10.992,149.494
C00596=1122.085,354.202,-83.788,-177.216,10.995,149.494
C00597=1122.081,354.449,-83.823,-177.212,10.997,149.494
C00598=1122.077,354.696,-83.858,-177.209,11.000,149.493
C00599=1122.073,354.944,-83.894,-177.205,11.002,149.493
C00600=1122.070,355.191,-83.929,-177.202,11.005,149.493
C00601=1122.065,355.439,-83.966,-177.199,11.007,149.493
C00602=1122.062,355.686,-84.001,-177.195,11.009,149.492
C00603=1122.058,355.934,-84.037,-177.192,11.012,149.492
C00604=1122.054,356.181,-84.072,-177.188,11.014,149.492
C00605=1122.050,356.428,-84.107,-177.184,11.018,149.492
C00606=1122.047,356.675,-84.144,-177.181,11.020,149.491
C00607=1122.042,356.923,-84.180,-177.177,11.022,149.491
C00608=1122.039,357.170,-84.215,-177.174,11.025,149.491
C00609=1122.035,357.418,-84.251,-177.171,11.027,149.491
C00610=1122.031,357.665,-84.286,-177.167,11.029,149.490
C00611=1122.028,357.913,-84.322,-177.164,11.032,149.490
C00612=1122.024,358.160,-84.359,-177.160,11.034,149.490
C00613=1122.020,358.408,-84.394,-177.157,11.037,149.490
C00614=1122.016,358.655,-84.430,-177.154,11.039,149.489
C00615=1122.013,358.903,-84.465,-177.150,11.041,149.489
C00616=1122.008,359.150,-84.501,-177.147,11.044,149.489
C00617=1122.004,359.397,-84.537,-177.143,11.046,149.488
C00618=1122.001,359.644,-84.573,-177.140,11.049,149.488
C00619=1121.996,359.892,-84.609,-177.136,11.051,149.488
C00620=1121.993,360.139,-84.645,-177.133,11.053,149.488
C00621=1121.989,360.386,-84.681,-177.130,11.056,149.487
C00622=1121.985,360.634,-84.717,-177.127,11.058,149.487
C00623=1121.981,360.881,-84.753,-177.123,11.060,149.487
C00624=1121.978,361.128,-84.789,-177.120,11.063,149.487
C00625=1121.974,361.376,-84.824,-177.116,11.065,149.486
C00626=1121.971,361.589,-84.856,-177.113,11.068,149.486
C00627=1121.967,361.801,-84.887,-177.110,11.069,149.486
C00628=1121.964,362.013,-84.918,-177.107,11.072,149.486
C00629=1121.961,362.225,-84.949,-177.104,11.074,149.485
C00630=1121.958,362.438,-84.980,-177.102,11.076,149.485
C00631=1121.954,362.650,-85.011,-177.099,11.078,149.485
C00632=1121.951,362.862,-85.042,-177.096,11.080,149.485
C00633=1121.948,363.075,-85.074,-177.093,11.082,149.485
C00634=1121.944,363.323,-85.109,-177.089,11.085,149.484
C00635=1121.941,363.569,-85.145,-177.086,11.087,149.484
C00636=1121.937,363.817,-85.182,-177.083,11.089,149.484
C00637=1121.933,364.064,-85.218,-177.080,11.091,149.484
C00638=1121.929,364.311,-85.255,-177.076,11.094,149.483
C00639=1121.925,364.559,-85.290,-177.073,11.096,149.483
C00640=1121.921,364.806,-85.327,-177.070,11.098,149.483
C00641=1121.918,365.053,-85.363,-177.066,11.101,149.483
C00642=1121.914,365.301,-85.399,-177.063,11.103,149.482
C00643=1121.910,365.548,-85.436,-177.059,11.106,149.482
C00644=1121.906,365.795,-85.472,-177.056,11.108,149.482
C00645=1121.902,366.042,-85.508,-177.053,11.111,149.482
C00646=1121.898,366.289,-85.545,-177.050,11.113,149.482
C00647=1121.895,366.538,-85.581,-177.046,11.115,149.481
C00648=1121.891,366.785,-85.618,-177.043,11.118,149.481
C00649=1121.888,367.032,-85.654,-177.040,11.119,149.481
C00650=1121.884,367.279,-85.691,-177.037,11.122,149.480
C00651=1121.879,367.527,-85.727,-177.033,11.124,149.480
C00652=1121.876,367.774,-85.763,-177.030,11.127,149.480
C00653=1121.872,368.021,-85.800,-177.027,11.129,149.480
C00654=1121.868,368.268,-85.836,-177.023,11.132,149.480
C00655=1121.864,368.515,-85.873,-177.020,11.134,149.479
C00656=1121.861,368.763,-85.910,-177.016,11.136,149.479
C00657=1121.857,369.010,-85.946,-177.013,11.139,149.479
C00658=1121.853,369.257,-85.983,-177.010,11.140,149.479
C00659=1121.850,369.504,-86.019,-177.007,11.143,149.478
C00660=1121.846,369.752,-86.056,-177.004,11.145,149.478
C00661=1121.842,369.999,-86.093,-177.001,11.148,149.478
C00662=1121.839,370.246,-86.130,-176.997,11.150,149.478
C00663=1121.835,370.493,-86.166,-176.994,11.153,149.478
C00664=1121.831,370.741,-86.203,-176.991,11.155,149.477
C00665=1121.826,370.988,-86.239,-176.987,11.158,149.477
C00666=1121.823,371.235,-86.276,-176.985,11.159,149.477
C00667=1121.819,371.483,-86.313,-176.981,11.162,149.477
C00668=1121.815,371.730,-86.350,-176.978,11.164,149.476
C00669=1121.812,371.977,-86.386,-176.975,11.167,149.476
C00670=1121.808,372.225,-86.423,-176.971,11.169,149.476
C00671=1121.804,372.471,-86.460,-176.968,11.172,149.476
C00672=1121.801,372.719,-86.498,-176.965,11.174,149.476
C00673=1121.797,372.966,-86.534,-176.962,11.176,149.475
C00674=1121.793,373.213,-86.571,-176.959,11.179,149.475
C00675=1121.789,373.460,-86.608,-176.956,11.181,149.475
C00676=1121.786,373.708,-86.645,-176.953,11.184,149.475
C00677=1121.781,373.955,-86.682,-176.949,11.186,149.475
C00678=1121.778,374.202,-86.718,-176.947,11.188,149.474
C00679=1121.774,374.449,-86.755,-176.943,11.190,149.474
C00680=1121.771,374.697,-86.793,-176.940,11.193,149.474
C00681=1121.767,374.944,-86.830,-176.937,11.195,149.474
C00682=1121.764,375.156,-86.861,-176.935,11.197,149.474
C00683=1121.761,375.369,-86.893,-176.932,11.199,149.474
C00684=1121.757,375.580,-86.925,-176.929,11.202,149.474
C00685=1121.754,375.793,-86.956,-176.926,11.204,149.473
C00686=1121.751,376.005,-86.988,-176.924,11.206,149.473
C00687=1121.748,376.217,-87.021,-176.921,11.208,149.473
C00688=1121.744,376.429,-87.052,-176.918,11.210,149.473
C00689=1121.741,376.641,-87.084,-176.916,11.212,149.473
C00690=1121.737,376.888,-87.121,-176.913,11.214,149.473
C00691=1121.734,377.136,-87.158,-176.910,11.217,149.473
C00692=1121.730,377.383,-87.196,-176.906,11.220,149.472
C00693=1121.726,377.630,-87.232,-176.904,11.221,149.472
C00694=1121.722,377.878,-87.270,-176.900,11.224,149.472
C00695=1121.718,378.124,-87.307,-176.897,11.227,149.472
C00696=1121.714,378.372,-87.344,-176.894,11.229,149.472
C00697=1121.711,378.619,-87.382,-176.891,11.232,149.471
C00698=1121.707,378.866,-87.419,-176.889,11.234,149.471
C00699=1121.703,379.113,-87.456,-176.885,11.236,149.471
C00700=1121.700,379.361,-87.494,-176.882,11.239,149.471
C00701=1121.696,379.608,-87.530,-176.879,11.241,149.471
C00702=1121.693,379.855,-87.568,-176.876,11.244,149.471
C00703=1121.688,380.102,-87.605,-176.874,11.246,149.471
C00704=1121.685,380.349,-87.643,-176.870,11.248,149.471
C00705=1121.681,380.597,-87.680,-176.867,11.251,149.471
C00706=1121.677,380.843,-87.718,-176.864,11.254,149.470
C00707=1121.673,381.090,-87.755,-176.861,11.257,149.470
C00708=1121.670,381.338,-87.792,-176.859,11.258,149.470
C00709=1121.666,381.585,-87.829,-176.856,11.261,149.470
C00710=1121.663,381.832,-87.867,-176.853,11.264,149.470
C00711=1121.659,382.079,-87.905,-176.849,11.266,149.470
C00712=1121.655,382.327,-87.942,-176.847,11.269,149.470
C00713=1121.652,382.573,-87.980,-176.844,11.271,149.470
C00714=1121.648,382.820,-88.016,-176.841,11.274,149.470
C00715=1121.644,383.068,-88.054,-176.838,11.277,149.470
C00716=1121.640,383.315,-88.093,-176.835,11.279,149.469
C00717=1121.636,383.562,-88.130,-176.832,11.281,149.469
C00718=1121.633,383.809,-88.167,-176.831,11.283,149.469
C00719=1121.629,384.056,-88.205,-176.828,11.285,149.469
C00720=1121.625,384.303,-88.242,-176.826,11.288,149.470
C00721=1121.622,384.551,-88.280,-176.825,11.289,149.469
C00722=1121.618,384.797,-88.318,-176.823,11.291,149.470
C00723=1121.614,385.045,-88.356,-176.821,11.294,149.470
C00724=1121.610,385.292,-88.393,-176.819,11.296,149.470
C00725=1121.607,385.539,-88.431,-176.817,11.298,149.470
C00726=1121.603,385.786,-88.469,-176.815,11.301,149.470
C00727=1121.600,386.033,-88.507,-176.813,11.303,149.470
C00728=1121.596,386.280,-88.543,-176.811,11.305,149.470
C00729=1121.592,386.528,-88.582,-176.809,11.307,149.470
C00730=1121.588,386.775,-88.620,-176.808,11.309,149.470
C00731=1121.585,387.022,-88.657,-176.806,11.311,149.470
C00732=1121.581,387.268,-88.695,-176.804,11.314,149.471
C00733=1121.578,387.516,-88.733,-176.802,11.316,149.471
C00734=1121.573,387.763,-88.770,-176.800,11.318,149.471
C00735=1121.570,388.010,-88.808,-176.798,11.321,149.471
C00736=1121.566,388.257,-88.846,-176.797,11.323,149.471
C00737=1121.563,388.504,-88.884,-176.795,11.325,149.471
C00738=1121.560,388.717,-88.916,-176.793,11.328,149.472
C00739=1121.557,388.929,-88.948,-176.792,11.330,149.472
C00740=1121.554,389.140,-88.982,-176.790,11.332,149.472
C00741=1121.550,389.353,-89.014,-176.789,11.334,149.472
C00742=1121.547,389.564,-89.046,-176.787,11.336,149.472
C00743=1121.544,389.776,-89.079,-176.785,11.339,149.472
C00744=1121.541,389.988,-89.111,-176.784,11.340,149.472
C00745=1121.538,390.200,-89.144,-176.783,11.343,149.473
C00746=1121.534,390.447,-89.182,-176.781,11.345,149.473
C00747=1121.530,390.694,-89.220,-176.779,11.348,149.473
C00748=1121.527,390.942,-89.258,-176.778,11.351,149.473
C00749=1121.524,391.189,-89.296,-176.776,11.353,149.474
C00750=1121.519,391.436,-89.334,-176.775,11.356,149.474
C00751=1121.516,391.683,-89.372,-176.773,11.358,149.474
C00752=1121.512,391.929,-89.410,-176.771,11.361,149.474
C00753=1121.509,392.177,-89.447,-176.769,11.364,149.475
C00754=1121.505,392.424,-89.486,-176.768,11.367,149.475
C00755=1121.501,392.671,-89.524,-176.766,11.370,149.475
C00756=1121.498,392.918,-89.562,-176.765,11.372,149.476
C00757=1121.493,393.165,-89.600,-176.763,11.375,149.476
C00758=1121.490,393.412,-89.638,-176.762,11.378,149.476
C00759=1121.486,393.660,-89.676,-176.760,11.380,149.477
C00760=1121.483,393.906,-89.714,-176.758,11.384,149.477
C00761=1121.479,394.154,-89.752,-176.757,11.387,149.478
C00762=1121.475,394.401,-89.790,-176.755,11.389,149.478
C00763=1121.472,394.648,-89.828,-176.754,11.392,149.478
C00764=1121.469,394.895,-89.866,-176.753,11.395,149.479
C00765=1121.464,395.141,-89.905,-176.751,11.399,149.479
C00766=1121.461,395.389,-89.943,-176.750,11.402,149.480
C00767=1121.457,395.636,-89.981,-176.748,11.404,149.480
C00768=1121.453,395.883,-90.019,-176.747,11.408,149.480
C00769=1121.449,396.130,-90.057,-176.745,11.411,149.481
C00770=1121.446,396.376,-90.095,-176.744,11.414,149.481
C00771=1121.443,396.624,-90.133,-176.743,11.417,149.482
C00772=1121.439,396.871,-90.172,-176.741,11.420,149.482
C00773=1121.435,397.118,-90.210,-176.740,11.423,149.483
C00774=1121.431,397.365,-90.248,-176.739,11.426,149.483
C00775=1121.428,397.612,-90.287,-176.737,11.430,149.484
C00776=1121.424,397.859,-90.325,-176.736,11.433,149.484
C00777=1121.420,398.106,-90.363,-176.735,11.436,149.485
C00778=1121.417,398.354,-90.401,-176.733,11.440,149.485
C00779=1121.413,398.600,-90.440,-176.732,11.443,149.486
C00780=1121.409,398.847,-90.478,-176.730,11.447,149.486
C00781=1121.406,399.095,-90.516,-176.729,11.450,149.487
C00782=1121.402,399.341,-90.555,-176.728,11.454,149.488
C00783=1121.399,399.588,-90.593,-176.727,11.457,149.488
C00784=1121.395,399.836,-90.631,-176.726,11.460,149.489
C00785=1121.391,400.082,-90.670,-176.724,11.464,149.489
C00786=1121.387,400.329,-90.708,-176.724,11.467,149.490
C00787=1121.384,400.577,-90.746,-176.722,11.471,149.491
C00788=1121.380,400.823,-90.785,-176.721,11.474,149.491
C00789=1121.377,401.070,-90.823,-176.720,11.479,149.492
C00790=1121.373,401.318,-90.862,-176.719,11.482,149.493
C00791=1121.370,401.564,-90.900,-176.717,11.486,149.493
C00792=1121.366,401.812,-90.939,-176.716,11.490,149.494
C00793=1121.362,402.058,-90.977,-176.715,11.493,149.495
C00794=1121.359,402.270,-91.010,-176.714,11.496,149.495
C00795=1121.356,402.482,-91.043,-176.714,11.500,149.496
C00796=1121.353,402.694,-91.076,-176.713,11.503,149.497
C00797=1121.350,402.906,-91.110,-176.712,11.506,149.497
C00798=1121.347,403.118,-91.143,-176.710,11.510,149.498
C00799=1121.343,403.330,-91.176,-176.710,11.513,149.499
C00800=1121.341,403.541,-91.209,-176.709,11.517,149.499
C00801=1121.337,403.754,-91.241,-176.708,11.520,149.500
C00802=1121.334,404.001,-91.280,-176.707,11.524,149.501
C00803=1121.330,404.247,-91.319,-176.706,11.528,149.501
C00804=1121.326,404.494,-91.357,-176.705,11.532,149.502
C00805=1121.323,404.741,-91.396,-176.704,11.536,149.503
C00806=1121.320,404.989,-91.434,-176.704,11.540,149.504
C00807=1121.315,405.235,-91.473,-176.703,11.544,149.505
C00808=1121.312,405.482,-91.512,-176.701,11.548,149.506
C00809=1121.309,405.729,-91.550,-176.700,11.553,149.507
C00810=1121.305,405.977,-91.589,-176.700,11.557,149.507
C00811=1121.301,406.224,-91.628,-176.699,11.561,149.508
C00812=1121.298,406.469,-91.667,-176.698,11.565,149.509
C00813=1121.294,406.717,-91.705,-176.697,11.570,149.510
C00814=1121.290,406.964,-91.744,-176.696,11.574,149.511
C00815=1121.287,407.211,-91.783,-176.695,11.579,149.512
C00816=1121.283,407.458,-91.822,-176.695,11.583,149.513
C00817=1121.280,407.705,-91.861,-176.695,11.587,149.514
C00818=1121.276,407.951,-91.899,-176.694,11.592,149.515
C00819=1121.272,408.199,-91.938,-176.693,11.596,149.516
C00820=1121.269,408.446,-91.977,-176.692,11.601,149.517
C00821=1121.266,408.692,-92.015,-176.692,11.606,149.518
C00822=1121.262,408.940,-92.054,-176.691,11.610,149.519
C00823=1121.258,409.187,-92.093,-176.690,11.615,149.520
C00824=1121.254,409.433,-92.132,-176.689,11.620,149.521
C00825=1121.251,409.680,-92.170,-176.689,11.624,149.522
C00826=1121.247,409.927,-92.209,-176.688,11.629,149.523
C00827=1121.244,410.174,-92.249,-176.688,11.634,149.524
C00828=1121.240,410.421,-92.288,-176.687,11.639,149.526
C00829=1121.237,410.668,-92.327,-176.687,11.643,149.527
C00830=1121.233,410.916,-92.365,-176.686,11.648,149.528
C00831=1121.229,411.162,-92.404,-176.685,11.653,149.529
C00832=1121.225,411.409,-92.443,-176.685,11.658,149.530
C00833=1121.222,411.656,-92.482,-176.684,11.664,149.531
C00834=1121.219,411.902,-92.521,-176.684,11.668,149.532
C00835=1121.215,412.149,-92.560,-176.683,11.673,149.534
C00836=1121.211,412.397,-92.599,-176.683,11.678,149.535
C00837=1121.208,412.644,-92.638,-176.683,11.683,149.536
C00838=1121.204,412.891,-92.677,-176.682,11.688,149.537
C00839=1121.201,413.138,-92.716,-176.681,11.694,149.539
C00840=1121.197,413.384,-92.755,-176.681,11.699,149.540
C00841=1121.193,413.631,-92.794,-176.681,11.704,149.541
C00842=1121.190,413.878,-92.833,-176.681,11.709,149.542
C00843=1121.187,414.125,-92.872,-176.680,11.715,149.544
C00844=1121.184,414.372,-92.911,-176.680,11.721,149.545
C00845=1121.183,414.619,-92.950,-176.680,11.726,149.546
C00846=1121.182,414.866,-92.989,-176.680,11.731,149.548
C00847=1121.181,415.113,-93.027,-176.679,11.737,149.549
C00848=1121.181,415.360,-93.066,-176.679,11.742,149.551
C00849=1121.182,415.606,-93.105,-176.679,11.747,149.552
C00850=1121.183,415.818,-93.138,-176.679,11.752,149.553
C00851=1121.183,416.030,-93.171,-176.678,11.757,149.554
C00852=1121.185,416.242,-93.204,-176.679,11.762,149.556
C00853=1121.187,416.454,-93.236,-176.679,11.767,149.557
C00854=1121.190,416.665,-93.269,-176.679,11.772,149.558
C00855=1121.192,416.877,-93.302,-176.678,11.777,149.560
C00856=1121.196,417.088,-93.335,-176.679,11.781,149.561
C00857=1121.200,417.301,-93.367,-176.679,11.786,149.562
C00858=1120.780,417.299,-93.430,-176.671,11.791,149.561
C00859=1120.777,417.088,-93.397,-176.671,11.786,149.560
C00860=1120.774,416.877,-93.364,-176.671,11.781,149.559
C00861=1120.771,416.665,-93.332,-176.671,11.776,149.558
C00862=1120.768,416.453,-93.299,-176.671,11.771,149.556
C00863=1120.766,416.242,-93.266,-176.672,11.766,149.555
C00864=1120.764,416.030,-93.234,-176.671,11.762,149.554
C00865=1120.763,415.818,-93.200,-176.672,11.757,149.553
C00866=1120.763,415.606,-93.167,-176.672,11.752,149.551
C00867=1120.762,415.360,-93.129,-176.672,11.747,149.550
C00868=1120.762,415.113,-93.090,-176.673,11.740,149.549
C00869=1120.763,414.865,-93.051,-176.673,11.735,149.547
C00870=1120.764,414.619,-93.012,-176.672,11.730,149.546
C00871=1120.766,414.372,-92.974,-176.673,11.724,149.544
C00872=1120.768,414.124,-92.935,-176.674,11.719,149.543
C00873=1120.770,413.878,-92.895,-176.674,11.714,149.542
C00874=1120.774,413.631,-92.856,-176.675,11.708,149.541
C00875=1120.778,413.384,-92.818,-176.675,11.703,149.539
C00876=1120.782,413.137,-92.778,-176.675,11.698,149.538
C00877=1120.785,412.890,-92.739,-176.676,11.692,149.537
C00878=1120.788,412.643,-92.700,-176.676,11.687,149.536
C00879=1120.792,412.396,-92.661,-176.676,11.682,149.534
C00880=1120.795,412.149,-92.622,-176.677,11.677,149.533
C00881=1120.800,411.903,-92.583,-176.678,11.671,149.532
C00882=1120.803,411.656,-92.544,-176.678,11.667,149.531
C00883=1120.806,411.409,-92.505,-176.679,11.662,149.530
C00884=1120.810,411.162,-92.467,-176.679,11.657,149.528
C00885=1120.814,410.915,-92.427,-176.680,11.652,149.527
C00886=1120.817,410.668,-92.388,-176.680,11.647,149.526
C00887=1120.821,410.421,-92.349,-176.681,11.642,149.525
C00888=1120.824,410.174,-92.310,-176.682,11.637,149.524
C00889=1120.827,409.927,-92.271,-176.683,11.632,149.523
C00890=1120.832,409.680,-92.233,-176.683,11.627,149.522
C00891=1120.835,409.433,-92.194,-176.684,11.623,149.521
C00892=1120.838,409.187,-92.155,-176.685,11.618,149.520
C00893=1120.842,408.940,-92.116,-176.685,11.613,149.518
C00894=1120.846,408.692,-92.077,-176.686,11.609,149.517
C00895=1120.849,408.445,-92.038,-176.687,11.604,149.516
C00896=1120.852,408.199,-91.999,-176.687,11.599,149.515
C00897=1120.857,407.952,-91.961,-176.688,11.595,149.514
C00898=1120.861,407.705,-91.922,-176.689,11.590,149.514
C00899=1120.863,407.458,-91.883,-176.690,11.586,149.512
C00900=1120.867,407.211,-91.844,-176.691,11.581,149.511
C00901=1120.871,406.964,-91.805,-176.692,11.577,149.511
C00902=1120.874,406.718,-91.767,-176.693,11.572,149.510
C00903=1120.878,406.470,-91.729,-176.693,11.569,149.509
C00904=1120.882,406.223,-91.689,-176.694,11.564,149.508
C00905=1120.885,405.976,-91.651,-176.695,11.560,149.507
C00906=1120.889,405.729,-91.612,-176.696,11.555,149.506
C00907=1120.892,405.482,-91.573,-176.697,11.551,149.505
C00908=1120.896,405.236,-91.535,-176.698,11.547,149.504
C00909=1120.900,404.988,-91.496,-176.698,11.543,149.503
C00910=1120.903,404.741,-91.457,-176.700,11.539,149.503
C00911=1120.907,404.494,-91.419,-176.701,11.535,149.502
C00912=1120.911,404.248,-91.380,-176.702,11.530,149.501
C00913=1120.915,404.000,-91.341,-176.703,11.526,149.500
C00914=1120.918,403.754,-91.303,-176.704,11.523,149.499
C00915=1120.921,403.542,-91.269,-176.704,11.519,149.499
C00916=1120.924,403.330,-91.237,-176.706,11.515,149.498
C00917=1120.927,403.118,-91.204,-176.707,11.512,149.498
C00918=1120.931,402.906,-91.170,-176.707,11.509,149.497
C00919=1120.934,402.694,-91.137,-176.708,11.506,149.496
C00920=1120.937,402.482,-91.105,-176.709,11.503,149.496
C00921=1120.940,402.271,-91.072,-176.710,11.499,149.495
C00922=1120.942,402.058,-91.038,-176.711,11.496,149.494
C00923=1120.947,401.811,-91.000,-176.712,11.492,149.494
C00924=1120.950,401.565,-90.961,-176.714,11.488,149.493
C00925=1120.954,401.317,-90.923,-176.714,11.485,149.492
C00926=1120.957,401.071,-90.884,-176.716,11.480,149.492
C00927=1120.961,400.824,-90.846,-176.717,11.477,149.491
C00928=1120.964,400.576,-90.808,-176.718,11.473,149.490
C00929=1120.968,400.329,-90.769,-176.720,11.470,149.490
C00930=1120.972,400.083,-90.731,-176.721,11.466,149.489
C00931=1120.976,399.835,-90.693,-176.722,11.462,149.488
C00932=1120.978,399.589,-90.654,-176.723,11.459,149.488
C00933=1120.983,399.342,-90.616,-176.725,11.455,149.487
C00934=1120.987,399.094,-90.577,-176.726,11.452,149.487
C00935=1120.990,398.848,-90.539,-176.727,11.448,149.486
C00936=1120.994,398.600,-90.500,-176.728,11.445,149.485
C00937=1120.997,398.353,-90.462,-176.729,11.442,149.485
C00938=1121.000,398.107,-90.424,-176.731,11.438,149.484
C00939=1121.004,397.859,-90.385,-176.732,11.435,149.484
C00940=1121.008,397.613,-90.348,-176.734,11.431,149.483
C00941=1121.012,397.365,-90.309,-176.735,11.429,149.483
C00942=1121.015,397.118,-90.270,-176.737,11.425,149.482
C00943=1121.019,396.871,-90.232,-176.738,11.422,149.482
C00944=1121.023,396.624,-90.194,-176.739,11.419,149.481
C00945=1121.026,396.377,-90.156,-176.741,11.415,149.481
C00946=1121.030,396.131,-90.118,-176.742,11.412,149.481
C00947=1121.034,395.883,-90.079,-176.743,11.409,149.480
C00948=1121.038,395.637,-90.041,-176.746,11.406,149.480
C00949=1121.041,395.389,-90.003,-176.747,11.403,149.479
C00950=1121.045,395.142,-89.965,-176.748,11.400,149.479
C00951=1121.049,394.895,-89.927,-176.750,11.397,149.478
C00952=1121.052,394.648,-89.888,-176.751,11.394,149.478
C00953=1121.055,394.401,-89.850,-176.753,11.391,149.478
C00954=1121.059,394.154,-89.813,-176.754,11.388,149.477
C00955=1121.063,393.907,-89.774,-176.756,11.385,149.477
C00956=1121.067,393.660,-89.737,-176.758,11.382,149.476
C00957=1121.071,393.413,-89.698,-176.759,11.379,149.476
C00958=1121.074,393.165,-89.660,-176.760,11.377,149.476
C00959=1121.078,392.919,-89.622,-176.762,11.374,149.475
C00960=1121.082,392.671,-89.584,-176.764,11.370,149.475
C00961=1121.086,392.425,-89.546,-176.766,11.368,149.475
C00962=1121.089,392.177,-89.508,-176.767,11.365,149.474
C00963=1121.093,391.930,-89.470,-176.769,11.363,149.474
C00964=1121.096,391.683,-89.432,-176.770,11.360,149.474
C00965=1121.100,391.436,-89.394,-176.772,11.357,149.474
C00966=1121.104,391.189,-89.356,-176.774,11.354,149.474
C00967=1121.107,390.942,-89.318,-176.776,11.352,149.473
C00968=1121.110,390.694,-89.280,-176.777,11.349,149.473
C00969=1121.114,390.448,-89.243,-176.779,11.346,149.473
C00970=1121.118,390.200,-89.204,-176.781,11.344,149.472
C00971=1121.121,389.989,-89.171,-176.783,11.341,149.472
C00972=1121.124,389.777,-89.139,-176.784,11.340,149.472
C00973=1121.128,389.564,-89.106,-176.785,11.337,149.472
C00974=1121.131,389.353,-89.075,-176.787,11.335,149.472
C00975=1121.134,389.141,-89.041,-176.788,11.333,149.472
C00976=1121.137,388.929,-89.009,-176.790,11.331,149.471
C00977=1121.140,388.717,-88.977,-176.791,11.329,149.471
C00978=1121.144,388.504,-88.944,-176.793,11.327,149.471
C00979=1121.147,388.257,-88.906,-176.795,11.324,149.471
C00980=1121.151,388.011,-88.869,-176.797,11.322,149.471
C00981=1121.154,387.763,-88.831,-176.799,11.320,149.471
C00982=1121.158,387.517,-88.793,-176.801,11.317,149.471
C00983=1121.162,387.269,-88.755,-176.802,11.315,149.470
C00984=1121.166,387.022,-88.718,-176.804,11.312,149.470
C00985=1121.169,386.775,-88.680,-176.806,11.310,149.470
C00986=1121.173,386.528,-88.642,-176.808,11.308,149.470
C00987=1121.176,386.281,-88.604,-176.810,11.305,149.470
C00988=1121.180,386.034,-88.566,-176.812,11.303,149.470
C00989=1121.184,385.786,-88.529,-176.814,11.301,149.470
C00990=1121.188,385.540,-88.491,-176.816,11.299,149.470
C00991=1121.191,385.292,-88.453,-176.818,11.296,149.470
C00992=1121.195,385.046,-88.416,-176.819,11.295,149.470
C00993=1121.198,384.798,-88.379,-176.821,11.293,149.470
C00994=1121.203,384.551,-88.340,-176.823,11.290,149.469
C00995=1121.206,384.304,-88.303,-176.825,11.288,149.469
C00996=1121.210,384.057,-88.265,-176.827,11.286,149.469
C00997=1121.213,383.809,-88.228,-176.830,11.284,149.469
C00998=1121.217,383.563,-88.190,-176.832,11.282,149.469
C00999=1121.220,383.315,-88.152,-176.834,11.279,149.469
C01000=1121.224,383.068,-88.115,-176.837,11.277,149.469
C01001=1121.227,382.821,-88.077,-176.840,11.274,149.469
C01002=1121.232,382.574,-88.039,-176.843,11.272,149.470
C01003=1121.236,382.327,-88.002,-176.846,11.270,149.470
C01004=1121.239,382.080,-87.964,-176.848,11.267,149.470
C01005=1121.243,381.832,-87.928,-176.852,11.264,149.470
C01006=1121.247,381.585,-87.890,-176.855,11.262,149.470
C01007=1121.250,381.339,-87.852,-176.858,11.259,149.470
C01008=1121.254,381.091,-87.815,-176.860,11.257,149.470
C01009=1121.258,380.844,-87.777,-176.863,11.255,149.470
C01010=1121.262,380.597,-87.740,-176.866,11.252,149.470
C01011=1121.265,380.350,-87.702,-176.870,11.249,149.471
C01012=1121.269,380.102,-87.666,-176.873,11.246,149.471
C01013=1121.273,379.856,-87.628,-176.875,11.245,149.471
C01014=1121.276,379.608,-87.591,-176.878,11.242,149.471
C01015=1121.280,379.361,-87.553,-176.881,11.239,149.471
C01016=1121.284,379.114,-87.516,-176.885,11.237,149.471
C01017=1121.287,378.867,-87.478,-176.888,11.234,149.471
C01018=1121.291,378.620,-87.442,-176.891,11.232,149.471
C01019=1121.295,378.372,-87.404,-176.893,11.230,149.472
C01020=1121.299,378.125,-87.367,-176.896,11.227,149.472
C01021=1121.303,377.878,-87.330,-176.900,11.225,149.472
C01022=1121.306,377.630,-87.293,-176.903,11.222,149.472
C01023=1121.310,377.384,-87.255,-176.906,11.219,149.472
C01024=1121.314,377.136,-87.218,-176.909,11.218,149.472
C01025=1121.318,376.889,-87.181,-176.912,11.215,149.473
C01026=1121.321,376.642,-87.143,-176.915,11.212,149.473
C01027=1121.325,376.429,-87.112,-176.917,11.211,149.473
C01028=1121.328,376.218,-87.081,-176.920,11.208,149.473
C01029=1121.331,376.006,-87.048,-176.923,11.206,149.473
C01030=1121.334,375.793,-87.017,-176.925,11.204,149.473
C01031=1121.337,375.581,-86.985,-176.928,11.202,149.473
C01032=1121.340,375.370,-86.953,-176.931,11.200,149.474
C01033=1121.344,375.157,-86.921,-176.934,11.198,149.474
C01034=1121.347,374.945,-86.889,-176.936,11.196,149.474
C01035=1121.351,374.697,-86.852,-176.940,11.194,149.474
C01036=1121.355,374.450,-86.816,-176.942,11.191,149.474
C01037=1121.358,374.203,-86.779,-176.946,11.188,149.474
C01038=1121.362,373.956,-86.741,-176.949,11.186,149.475
C01039=1121.366,373.709,-86.704,-176.952,11.184,149.475
C01040=1121.370,373.462,-86.668,-176.955,11.182,149.475
C01041=1121.373,373.214,-86.630,-176.958,11.179,149.475
C01042=1121.377,372.967,-86.594,-176.962,11.177,149.475
C01043=1121.381,372.720,-86.557,-176.965,11.174,149.476
C01044=1121.385,372.473,-86.520,-176.968,11.172,149.476
C01045=1121.388,372.225,-86.483,-176.971,11.169,149.476
C01046=1121.392,371.978,-86.447,-176.974,11.168,149.476
C01047=1121.396,371.731,-86.410,-176.977,11.165,149.476
C01048=1121.400,371.483,-86.373,-176.981,11.163,149.477
C01049=1121.403,371.236,-86.336,-176.984,11.160,149.477
C01050=1121.407,370.989,-86.300,-176.987,11.158,149.477
C01051=1121.411,370.742,-86.263,-176.991,11.155,149.477
C01052=1121.415,370.494,-86.226,-176.994,11.153,149.478
C01053=1121.418,370.247,-86.190,-176.997,11.151,149.478
C01054=1121.422,370.000,-86.153,-177.000,11.149,149.478
C01055=1121.426,369.752,-86.116,-177.003,11.146,149.478
C01056=1121.429,369.505,-86.079,-177.007,11.144,149.478
C01057=1121.433,369.258,-86.043,-177.010,11.141,149.479
C01058=1121.438,369.010,-86.006,-177.013,11.139,149.479
C01059=1121.441,368.764,-85.970,-177.016,11.136,149.479
C01060=1121.445,368.516,-85.933,-177.020,11.134,149.479
C01061=1121.449,368.269,-85.896,-177.022,11.132,149.479
C01062=1121.452,368.022,-85.860,-177.026,11.130,149.480
C01063=1121.456,367.774,-85.823,-177.029,11.127,149.480
C01064=1121.460,367.527,-85.787,-177.033,11.125,149.480
C01065=1121.464,367.280,-85.751,-177.036,11.123,149.480
C01066=1121.467,367.033,-85.714,-177.039,11.120,149.481
C01067=1121.471,366.786,-85.677,-177.043,11.118,149.481
C01068=1121.476,366.538,-85.641,-177.046,11.115,149.481
C01069=1121.479,366.290,-85.605,-177.049,11.113,149.481
C01070=1121.483,366.043,-85.568,-177.052,11.110,149.482
C01071=1121.486,365.796,-85.532,-177.056,11.108,149.482
C01072=1121.490,365.548,-85.495,-177.059,11.106,149.482
C01073=1121.494,365.302,-85.459,-177.062,11.104,149.482
C01074=1121.498,365.054,-85.423,-177.065,11.101,149.483
C01075=1121.502,364.807,-85.387,-177.069,11.099,149.483
C01076=1121.506,364.559,-85.351,-177.072,11.096,149.483
C01077=1121.509,364.312,-85.314,-177.076,11.094,149.483
C01078=1121.513,364.065,-85.277,-177.079,11.092,149.484
C01079=1121.517,363.817,-85.242,-177.082,11.089,149.484
C01080=1121.521,363.570,-85.205,-177.086,11.087,149.484
C01081=1121.525,363.323,-85.169,-177.089,11.084,149.484
C01082=1121.528,363.076,-85.133,-177.092,11.082,149.484
C01083=1121.531,362.863,-85.102,-177.095,11.080,149.485
C01084=1121.535,362.651,-85.071,-177.098,11.078,149.485
C01085=1121.538,362.439,-85.040,-177.101,11.076,149.485
C01086=1121.541,362.226,-85.008,-177.104,11.074,149.485
C01087=1121.545,362.014,-84.978,-177.107,11.072,149.486
C01088=1121.548,361.801,-84.946,-177.110,11.070,149.486
C01089=1121.551,361.589,-84.917,-177.113,11.068,149.486
C01090=1121.554,361.376,-84.885,-177.116,11.066,149.486
C01091=1121.558,361.129,-84.849,-177.119,11.064,149.487
C01092=1121.562,360.882,-84.813,-177.122,11.061,149.487
C01093=1121.565,360.635,-84.777,-177.125,11.059,149.487
C01094=1121.569,360.387,-84.741,-177.129,11.057,149.487
C01095=1121.573,360.140,-84.705,-177.133,11.054,149.488
C01096=1121.576,359.893,-84.669,-177.136,11.052,149.488
C01097=1121.581,359.646,-84.633,-177.139,11.049,149.488
C01098=1121.585,359.398,-84.597,-177.142,11.047,149.488
C01099=1121.589,359.151,-84.562,-177.146,11.045,149.489
C01100=1121.592,358.904,-84.526,-177.149,11.042,149.489
C01101=1121.597,358.656,-84.490,-177.153,11.040,149.489
C01102=1121.600,358.408,-84.454,-177.156,11.037,149.489
C01103=1121.604,358.161,-84.418,-177.160,11.035,149.490
C01104=1121.607,357.914,-84.382,-177.163,11.033,149.490
C01105=1121.612,357.666,-84.346,-177.167,11.029,149.490
C01106=1121.615,357.419,-84.310,-177.170,11.027,149.490
C01107=1121.619,357.171,-84.275,-177.174,11.025,149.491
C01108=1121.623,356.924,-84.239,-177.177,11.022,149.491
C01109=1121.626,356.676,-84.204,-177.181,11.020,149.491
C01110=1121.631,356.429,-84.168,-177.184,11.017,149.491
C01111=1121.635,356.182,-84.132,-177.187,11.015,149.492
C01112=1121.638,355.935,-84.096,-177.191,11.013,149.492
C01113=1121.642,355.687,-84.061,-177.194,11.010,149.492
C01114=1121.646,355.440,-84.025,-177.198,11.008,149.493
C01115=1121.649,355.192,-83.990,-177.201,11.005,149.493
C01116=1121.654,354.944,-83.953,-177.205,11.002,149.493
C01117=1121.658,354.698,-83.918,-177.209,11.000,149.493
C01118=1121.662,354.450,-83.883,-177.212,10.997,149.494
C01119=1121.665,354.203,-83.847,-177.215,10.995,149.494
C01120=1121.669,353.955,-83.812,-177.218,10.993,149.494
C01121=1121.673,353.708,-83.776,-177.222,10.990,149.494
C01122=1121.676,353.460,-83.741,-177.225,10.988,149.495
C01123=1121.681,353.213,-83.706,-177.229,10.985,149.495
C01124=1121.684,352.965,-83.671,-177.233,10.982,149.495
C01125=1121.688,352.718,-83.635,-177.236,10.980,149.495
C01126=1121.692,352.470,-83.599,-177.239,10.977,149.496
C01127=1121.695,352.223,-83.564,-177.243,10.975,149.496
C01128=1121.700,351.976,-83.529,-177.246,10.973,149.496
C01129=1121.703,351.728,-83.493,-177.250,10.969,149.496
C01130=1121.707,351.480,-83.458,-177.254,10.967,149.497
C01131=1121.711,351.233,-83.423,-177.257,10.965,149.497
C01132=1121.715,350.986,-83.388,-177.260,10.962,149.497
C01133=1121.719,350.738,-83.352,-177.264,10.960,149.497
C01134=1121.723,350.490,-83.317,-177.268,10.957,149.498
C01135=1121.727,350.243,-83.282,-177.271,10.954,149.498
C01136=1121.731,349.996,-83.246,-177.274,10.952,149.498
C01137=1121.735,349.748,-83.212,-177.278,10.949,149.498
C01138=1121.738,349.500,-83.176,-177.282,10.946,149.498
C01139=1121.742,349.288,-83.146,-177.284,10.944,149.499
C01140=1121.745,349.076,-83.116,-177.287,10.942,149.499
C01141=1121.749,348.863,-83.085,-177.290,10.940,149.499
C01142=1121.752,348.651,-83.055,-177.293,10.938,149.499
C01143=1121.756,348.438,-83.025,-177.296,10.935,149.499
C01144=1121.759,348.226,-82.996,-177.298,10.934,149.500
C01145=1121.762,348.013,-82.964,-177.301,10.932,149.500
C01146=1121.765,347.801,-82.935,-177.304,10.929,149.500
C01147=1121.769,347.553,-82.900,-177.307,10.927,149.500
C01148=1121.774,347.306,-82.865,-177.311,10.924,149.500
C01149=1121.778,347.058,-82.830,-177.314,10.922,149.501
C01150=1121.780,346.811,-82.795,-177.316,10.920,149.501
C01151=1121.785,346.563,-82.760,-177.319,10.917,149.501
C01152=1121.789,346.316,-82.725,-177.323,10.915,149.501
C01153=1121.793,346.068,-82.690,-177.326,10.913,149.501
C01154=1121.797,345.821,-82.655,-177.329,10.910,149.502
C01155=1121.800,345.573,-82.621,-177.333,10.908,149.502
C01156=1121.804,345.326,-82.586,-177.336,10.905,149.502
C01157=1121.808,345.078,-82.551,-177.339,10.902,149.502
C01158=1121.812,344.831,-82.515,-177.342,10.900,149.502
C01159=1121.817,344.583,-82.481,-177.346,10.897,149.503
C01160=1121.820,344.335,-82.446,-177.349,10.895,149.503
C01161=1121.824,344.089,-82.411,-177.352,10.893,149.503
C01162=1121.828,343.841,-82.376,-177.355,10.890,149.503
C01163=1121.832,343.592,-82.342,-177.358,10.887,149.503
C01164=1121.836,343.346,-82.307,-177.362,10.885,149.504
C01165=1121.840,343.098,-82.272,-177.365,10.882,149.504
C01166=1121.844,342.850,-82.238,-177.368,10.881,149.504
C01167=1121.847,342.603,-82.203,-177.371,10.878,149.504
C01168=1121.852,342.356,-82.168,-177.374,10.875,149.504
C01169=1121.856,342.108,-82.133,-177.377,10.873,149.505
C01170=1121.860,341.860,-82.099,-177.381,10.871,149.505
C01171=1121.863,341.612,-82.065,-177.384,10.868,149.505
C01172=1121.868,341.366,-82.030,-177.387,10.866,149.505
C01173=1121.872,341.118,-81.995,-177.390,10.863,149.505
C01174=1121.875,340.870,-81.961,-177.393,10.860,149.506
C01175=1121.879,340.622,-81.926,-177.397,10.858,149.506
C01176=1121.883,340.374,-81.892,-177.400,10.855,149.506
C01177=1121.887,340.127,-81.857,-177.403,10.853,149.506
C01178=1121.892,339.880,-81.823,-177.406,10.850,149.506
C01179=1121.895,339.632,-81.789,-177.410,10.848,149.507
C01180=1121.899,339.385,-81.753,-177.413,10.845,149.507
C01181=1121.902,339.137,-81.719,-177.416,10.843,149.507
C01182=1121.907,338.890,-81.685,-177.419,10.841,149.507
C01183=1121.911,338.642,-81.650,-177.422,10.838,149.507
C01184=1121.915,338.395,-81.616,-177.425,10.836,149.508
C01185=1121.919,338.146,-81.581,-177.428,10.834,149.508
C01186=1121.923,337.899,-81.547,-177.432,10.831,149.508
C01187=1121.927,337.651,-81.512,-177.435,10.828,149.508
C01188=1121.930,337.404,-81.479,-177.438,10.826,149.508
C01189=1121.934,337.156,-81.444,-177.441,10.823,149.509
C01190=1121.938,336.909,-81.410,-177.445,10.821,149.509
C01191=1121.943,336.660,-81.376,-177.448,10.818,149.509
C01192=1121.946,336.413,-81.342,-177.451,10.816,149.509
C01193=1121.951,336.166,-81.307,-177.454,10.813,149.509
C01194=1121.954,335.918,-81.273,-177.458,10.811,149.510
C01195=1121.957,335.706,-81.244,-177.460,10.809,149.510
C01196=1121.961,335.493,-81.215,-177.463,10.807,149.510
C01197=1121.964,335.280,-81.185,-177.465,10.804,149.510
C01198=1121.968,335.068,-81.156,-177.468,10.803,149.510
C01199=1121.971,334.855,-81.127,-177.471,10.800,149.510
C01200=1121.974,334.642,-81.098,-177.474,10.798,149.511
C01201=1121.978,334.430,-81.068,-177.476,10.796,149.511
C01202=1121.982,334.217,-81.039,-177.479,10.794,149.511
C01203=1121.985,333.969,-81.004,-177.482,10.791,149.511
C01204=1121.989,333.722,-80.971,-177.486,10.788,149.511
C01205=1121.993,333.475,-80.936,-177.489,10.786,149.511
C01206=1121.997,333.226,-80.903,-177.492,10.784,149.512
C01207=1122.001,332.979,-80.869,-177.494,10.782,149.512
C01208=1122.005,332.732,-80.834,-177.498,10.779,149.512
C01209=1122.009,332.483,-80.801,-177.501,10.777,149.512
C01210=1122.013,332.236,-80.767,-177.504,10.774,149.512
C01211=1122.017,331.989,-80.732,-177.507,10.771,149.513
C01212=1122.021,331.740,-80.699,-177.511,10.769,149.513
C01213=1122.025,331.493,-80.665,-177.514,10.767,149.513
C01214=1122.029,331.246,-80.631,-177.517,10.764,149.513
C01215=1122.033,330.997,-80.597,-177.520,10.761,149.513
C01216=1122.037,330.750,-80.563,-177.524,10.759,149.514
C01217=1122.041,330.502,-80.530,-177.527,10.756,149.514
C01218=1122.044,330.255,-80.496,-177.530,10.754,149.514
C01219=1122.049,330.007,-80.462,-177.533,10.751,149.514
C01220=1122.053,329.759,-80.428,-177.536,10.749,149.514
C01221=1122.057,329.512,-80.395,-177.539,10.747,149.514
C01222=1122.060,329.264,-80.361,-177.542,10.744,149.515
C01223=1122.065,329.016,-80.327,-177.545,10.742,149.515
C01224=1122.069,328.769,-80.293,-177.549,10.739,149.515
C01225=1122.073,328.521,-80.260,-177.552,10.737,149.515
C01226=1122.076,328.273,-80.226,-177.555,10.734,149.515
C01227=1122.080,328.026,-80.193,-177.558,10.732,149.516
C01228=1122.085,327.778,-80.158,-177.561,10.729,149.516
C01229=1122.089,327.530,-80.125,-177.565,10.727,149.516
C01230=1122.093,327.282,-80.091,-177.568,10.724,149.516
C01231=1122.096,327.035,-80.058,-177.571,10.721,149.516
C01232=1122.101,326.787,-80.024,-177.574,10.719,149.517
C01233=1122.105,326.539,-79.991,-177.577,10.716,149.517
C01234=1122.108,326.292,-79.957,-177.580,10.714,149.517
C01235=1122.112,326.044,-79.924,-177.584,10.711,149.517
C01236=1122.116,325.796,-79.891,-177.586,10.710,149.517
C01237=1122.121,325.549,-79.856,-177.589,10.707,149.517
C01238=1122.125,325.301,-79.823,-177.593,10.704,149.518
C01239=1122.128,325.053,-79.790,-177.596,10.702,149.518
C01240=1122.133,324.805,-79.756,-177.599,10.699,149.518
C01241=1122.136,324.558,-79.723,-177.602,10.697,149.518
C01242=1122.141,324.310,-79.689,-177.605,10.694,149.519
C01243=1122.145,324.062,-79.656,-177.608,10.691,149.519
C01244=1122.149,323.815,-79.623,-177.612,10.689,149.519
C01245=1122.152,323.566,-79.590,-177.615,10.687,149.519
C01246=1122.156,323.319,-79.556,-177.618,10.684,149.519
C01247=1122.160,323.071,-79.523,-177.621,10.681,149.519
C01248=1122.164,322.824,-79.489,-177.625,10.679,149.520
C01249=1122.169,322.576,-79.456,-177.628,10.676,149.520
C01250=1122.173,322.328,-79.423,-177.630,10.674,149.520
C01251=1122.179,321.914,-79.368,-177.636,10.670,149.520
C01252=1122.185,321.502,-79.312,-177.641,10.666,149.521
C01253=1122.192,321.089,-79.257,-177.646,10.662,149.521
C01254=1122.199,320.676,-79.201,-177.652,10.657,149.521
C01255=1122.203,320.429,-79.169,-177.655,10.655,149.521
C01256=1122.207,320.181,-79.136,-177.658,10.652,149.522
C01257=1122.210,319.933,-79.102,-177.661,10.650,149.522
C01258=1122.215,319.684,-79.070,-177.664,10.648,149.522
C01259=1122.219,319.437,-79.037,-177.667,10.645,149.522
C01260=1122.223,319.189,-79.003,-177.670,10.643,149.522
C01261=1122.227,318.941,-78.970,-177.673,10.640,149.522
C01262=1122.231,318.694,-78.938,-177.676,10.637,149.523
C01263=1122.235,318.446,-78.904,-177.680,10.635,149.523
C01264=1122.239,318.198,-78.871,-177.683,10.632,149.523
C01265=1122.243,317.951,-78.838,-177.686,10.630,149.523
C01266=1122.247,317.703,-78.805,-177.689,10.627,149.524
C01267=1122.251,317.455,-78.773,-177.692,10.624,149.524
C01268=1122.255,317.207,-78.740,-177.696,10.622,149.524
C01269=1122.259,316.959,-78.707,-177.699,10.619,149.524
C01270=1122.263,316.712,-78.674,-177.702,10.617,149.524
C01271=1122.267,316.464,-78.642,-177.705,10.615,149.524
C01272=1122.271,316.216,-78.609,-177.708,10.612,149.525
C01273=1122.275,315.968,-78.576,-177.711,10.610,149.525
C01274=1122.279,315.720,-78.542,-177.714,10.607,149.525
C01275=1122.283,315.472,-78.511,-177.717,10.605,149.525
C01276=1122.287,315.225,-78.477,-177.720,10.602,149.525
C01277=1122.291,314.977,-78.444,-177.723,10.599,149.525
C01278=1122.295,314.729,-78.412,-177.727,10.597,149.526
C01279=1122.299,314.481,-78.379,-177.730,10.594,149.526
C01280=1122.303,314.233,-78.346,-177.733,10.592,149.526
C01281=1122.307,313.985,-78.314,-177.736,10.589,149.526
C01282=1122.311,313.738,-78.281,-177.739,10.587,149.526
C01283=1122.316,313.478,-78.247,-177.743,10.584,149.527
C01284=1122.320,313.217,-78.212,-177.746,10.582,149.527
C01285=1122.324,312.956,-78.179,-177.749,10.579,149.527
C01286=1122.329,312.696,-78.144,-177.752,10.577,149.527
C01287=1122.333,312.448,-78.111,-177.755,10.574,149.527
C01288=1122.336,312.200,-78.079,-177.758,10.571,149.527
C01289=1122.341,311.953,-78.046,-177.762,10.569,149.528
C01290=1122.344,311.705,-78.014,-177.765,10.566,149.528
C01291=1122.348,311.457,-77.981,-177.768,10.564,149.528
C01292=1122.353,311.210,-77.950,-177.771,10.561,149.528
C01293=1122.357,310.962,-77.917,-177.774,10.558,149.528
C01294=1122.361,310.714,-77.884,-177.777,10.557,149.529
C01295=1122.365,310.466,-77.852,-177.780,10.554,149.529
C01296=1122.369,310.218,-77.819,-177.783,10.552,149.529
C01297=1122.373,309.970,-77.787,-177.786,10.549,149.529
C01298=1122.377,309.722,-77.754,-177.789,10.546,149.529
C01299=1122.381,309.475,-77.723,-177.792,10.544,149.529
C01300=1122.386,309.226,-77.690,-177.796,10.541,149.530
C01301=1122.389,308.979,-77.658,-177.799,10.539,149.530
C01302=1122.394,308.731,-77.625,-177.802,10.536,149.530
C01303=1122.397,308.517,-77.598,-177.804,10.534,149.530
C01304=1122.400,308.305,-77.570,-177.808,10.532,149.530
C01305=1122.404,308.092,-77.542,-177.810,10.530,149.530
C01306=1122.408,307.880,-77.514,-177.812,10.528,149.531
C01307=1122.411,307.666,-77.487,-177.815,10.525,149.531
C01308=1122.414,307.453,-77.459,-177.818,10.523,149.531
C01309=1122.418,307.240,-77.431,-177.820,10.521,149.531
C01310=1122.421,307.027,-77.404,-177.823,10.519,149.531
C01311=1122.426,306.780,-77.372,-177.826,10.516,149.531
C01312=1122.430,306.531,-77.340,-177.830,10.514,149.532
C01313=1122.433,306.284,-77.307,-177.833,10.511,149.532
C01314=1122.438,306.036,-77.275,-177.835,10.509,149.532
C01315=1122.442,305.788,-77.243,-177.838,10.506,149.532
C01316=1122.446,305.540,-77.212,-177.842,10.504,149.532
C01317=1122.450,305.292,-77.179,-177.845,10.501,149.533
C01318=1122.454,305.044,-77.147,-177.848,10.499,149.533
C01319=1122.458,304.796,-77.115,-177.851,10.496,149.533
C01320=1122.462,304.549,-77.083,-177.854,10.493,149.533
C01321=1122.466,304.301,-77.051,-177.857,10.491,149.533
C01322=1122.470,304.053,-77.019,-177.860,10.488,149.533
C01323=1122.475,303.805,-76.987,-177.864,10.486,149.534
C01324=1122.479,303.557,-76.955,-177.867,10.483,149.534
C01325=1122.482,303.309,-76.923,-177.870,10.481,149.534
C01326=1122.487,303.061,-76.891,-177.872,10.479,149.534
C01327=1122.491,302.813,-76.859,-177.876,10.476,149.534
C01328=1122.495,302.565,-76.827,-177.879,10.473,149.534
C01329=1122.499,302.317,-76.795,-177.882,10.471,149.535
C01330=1122.504,302.070,-76.763,-177.885,10.468,149.535
C01331=1122.508,301.821,-76.732,-177.888,10.466,149.535
C01332=1122.511,301.573,-76.700,-177.891,10.463,149.535
C01333=1122.516,301.325,-76.668,-177.894,10.461,149.535
C01334=1122.520,301.077,-76.637,-177.897,10.458,149.535
C01335=1122.524,300.829,-76.605,-177.901,10.455,149.536
C01336=1122.528,300.582,-76.573,-177.904,10.453,149.536
C01337=1122.532,300.334,-76.541,-177.907,10.450,149.536
C01338=1122.537,300.086,-76.509,-177.910,10.449,149.536
C01339=1122.541,299.838,-76.478,-177.913,10.446,149.536
C01340=1122.544,299.589,-76.446,-177.916,10.443,149.537
C01341=1122.549,299.342,-76.415,-177.919,10.441,149.537
C01342=1122.552,299.094,-76.383,-177.922,10.438,149.537
C01343=1122.557,298.845,-76.352,-177.925,10.435,149.537
C01344=1122.561,298.598,-76.320,-177.928,10.433,149.537
C01345=1122.565,298.350,-76.288,-177.931,10.430,149.538
C01346=1122.570,298.102,-76.257,-177.935,10.428,149.538
C01347=1122.574,297.854,-76.225,-177.938,10.425,149.538
C01348=1122.577,297.606,-76.194,-177.941,10.423,149.538
C01349=1122.582,297.358,-76.162,-177.943,10.421,149.538
C01350=1122.586,297.110,-76.131,-177.947,10.418,149.539
C01351=1122.590,296.862,-76.099,-177.950,10.415,149.539
C01352=1122.594,296.614,-76.068,-177.952,10.413,149.539
C01353=1122.598,296.366,-76.037,-177.956,10.410,149.539
C01354=1122.602,296.118,-76.005,-177.959,10.407,149.539
C01355=1122.607,295.870,-75.974,-177.962,10.405,149.539
C01356=1122.610,295.622,-75.942,-177.965,10.402,149.539
C01357=1122.614,295.374,-75.911,-177.968,10.400,149.540
C01358=1122.619,295.126,-75.880,-177.971,10.397,149.540
C01359=1122.622,294.913,-75.852,-177.974,10.395,149.540
C01360=1122.626,294.700,-75.826,-177.976,10.393,149.540
C01361=1122.629,294.488,-75.798,-177.979,10.391,149.540
C01362=1122.633,294.274,-75.772,-177.981,10.389,149.540
C01363=1122.636,294.061,-75.744,-177.984,10.387,149.541
C01364=1122.640,293.848,-75.718,-177.987,10.384,149.541
C01365=1122.643,293.635,-75.692,-177.989,10.382,149.541
C01366=1122.647,293.422,-75.664,-177.992,10.381,149.541
C01367=1122.651,293.174,-75.633,-177.995,10.378,149.541
C01368=1122.655,292.926,-75.602,-177.998,10.375,149.541
C01369=1122.659,292.678,-75.571,-178.001,10.373,149.542
C01370=1122.664,292.430,-75.540,-178.004,10.370,149.542
C01371=1122.667,292.182,-75.508,-178.008,10.367,149.542
C01372=1122.672,291.934,-75.477,-178.011,10.365,149.542
C01373=1122.675,291.686,-75.446,-178.014,10.362,149.542
C01374=1122.680,291.438,-75.415,-178.017,10.360,149.542
C01375=1122.684,291.190,-75.385,-178.020,10.357,149.543
C01376=1122.688,290.942,-75.353,-178.023,10.354,149.543
C01377=1122.693,290.694,-75.322,-178.026,10.353,149.543
C01378=1122.697,290.445,-75.291,-178.029,10.350,149.543
C01379=1122.701,290.197,-75.260,-178.032,10.348,149.543
C01380=1122.704,289.950,-75.229,-178.035,10.345,149.544
C01381=1122.709,289.702,-75.198,-178.038,10.342,149.544
C01382=1122.713,289.453,-75.167,-178.041,10.340,149.544
C01383=1122.717,289.205,-75.136,-178.044,10.337,149.544
C01384=1122.721,288.958,-75.105,-178.048,10.334,149.544
C01385=1122.725,288.709,-75.074,-178.050,10.332,149.544
C01386=1122.730,288.461,-75.043,-178.054,10.329,149.545
C01387=1122.734,288.213,-75.013,-178.056,10.327,149.545
C01388=1122.737,287.965,-74.982,-178.059,10.325,149.545
C01389=1122.742,287.717,-74.951,-178.062,10.322,149.545
C01390=1122.746,287.469,-74.919,-178.065,10.319,149.545
C01391=1122.750,287.221,-74.889,-178.069,10.317,149.545
C01392=1122.754,286.973,-74.859,-178.072,10.314,149.546
C01393=1122.758,286.725,-74.827,-178.075,10.312,149.546
C01394=1122.763,286.477,-74.797,-178.078,10.309,149.546
C01395=1122.767,286.229,-74.766,-178.081,10.306,149.546
C01396=1122.771,285.981,-74.735,-178.084,10.304,149.546
C01397=1122.775,285.733,-74.705,-178.087,10.302,149.547
C01398=1122.779,285.485,-74.674,-178.090,10.299,149.547
C01399=1122.783,285.236,-74.643,-178.093,10.297,149.547
C01400=1122.788,284.988,-74.613,-178.096,10.294,149.547
C01401=1122.792,284.741,-74.582,-178.099,10.291,149.547
C01402=1122.796,284.492,-74.551,-178.102,10.289,149.547
C01403=1122.800,284.244,-74.520,-178.105,10.286,149.548
C01404=1122.804,283.996,-74.490,-178.109,10.284,149.548
C01405=1122.809,283.748,-74.460,-178.112,10.281,149.548
C01406=1122.812,283.500,-74.429,-178.114,10.279,149.548
C01407=1122.817,283.252,-74.399,-178.117,10.277,149.548
C01408=1122.822,283.004,-74.368,-178.120,10.274,149.548
C01409=1122.825,282.755,-74.338,-178.124,10.271,149.549
C01410=1122.830,282.507,-74.307,-178.126,10.269,149.549
C01411=1122.833,282.260,-74.277,-178.130,10.266,149.549
C01412=1122.838,282.012,-74.246,-178.133,10.263,149.549
C01413=1122.842,281.763,-74.216,-178.136,10.261,149.549
C01414=1122.846,281.515,-74.185,-178.139,10.258,149.550
C01415=1122.850,281.302,-74.159,-178.141,10.256,149.550
C01416=1122.854,281.089,-74.133,-178.145,10.254,149.550
C01417=1122.857,280.876,-74.107,-178.148,10.251,149.550
C01418=1122.861,280.662,-74.081,-178.150,10.249,149.550
C01419=1122.864,280.449,-74.055,-178.153,10.247,149.550
C01420=1122.868,280.236,-74.029,-178.156,10.244,149.551
C01421=1122.871,280.023,-74.003,-178.159,10.242,149.551
C01422=1122.875,279.809,-73.977,-178.162,10.240,149.551
C01423=1122.879,279.562,-73.947,-178.165,10.237,149.551
C01424=1122.884,279.314,-73.916,-178.168,10.234,149.551
C01425=1122.888,279.065,-73.886,-178.172,10.231,149.551
C01426=1122.892,278.817,-73.855,-178.175,10.228,149.552
C01427=1122.896,278.568,-73.826,-178.178,10.226,149.552
C01428=1122.900,278.321,-73.796,-178.181,10.223,149.552
C01429=1122.905,278.073,-73.765,-178.184,10.221,149.552
C01430=1122.909,277.824,-73.736,-178.188,10.218,149.552
C01431=1122.913,277.577,-73.705,-178.191,10.215,149.553
C01432=1122.917,277.328,-73.675,-178.194,10.212,149.553
C01433=1122.921,277.080,-73.645,-178.197,10.209,149.553
C01434=1122.925,276.832,-73.615,-178.200,10.207,149.553
C01435=1122.930,276.584,-73.585,-178.203,10.204,149.553
C01436=1122.934,276.335,-73.555,-178.207,10.201,149.553
C01437=1122.938,276.088,-73.525,-178.210,10.199,149.553
C01438=1122.943,275.839,-73.495,-178.213,10.196,149.554
C01439=1122.946,275.591,-73.464,-178.215,10.193,149.554
C01440=1122.950,275.343,-73.435,-178.219,10.191,149.554
C01441=1122.954,275.094,-73.405,-178.222,10.188,149.554
C01442=1122.959,274.846,-73.375,-178.225,10.185,149.554
C01443=1122.963,274.598,-73.345,-178.228,10.182,149.554
C01444=1122.967,274.350,-73.315,-178.231,10.180,149.555
C01445=1122.971,274.102,-73.286,-178.234,10.177,149.555
C01446=1122.976,273.854,-73.256,-178.237,10.175,149.555
C01447=1122.980,273.606,-73.225,-178.240,10.172,149.555
C01448=1122.984,273.358,-73.196,-178.243,10.169,149.555
C01449=1122.988,273.109,-73.166,-178.246,10.166,149.555
C01450=1122.992,272.862,-73.136,-178.249,10.164,149.555
C01451=1122.997,272.613,-73.106,-178.252,10.161,149.555
C01452=1123.001,272.365,-73.077,-178.255,10.158,149.556
C01453=1123.005,272.117,-73.047,-178.258,10.156,149.556
C01454=1123.010,271.868,-73.018,-178.261,10.153,149.556
C01455=1123.014,271.621,-72.988,-178.263,10.151,149.556
C01456=1123.018,271.372,-72.958,-178.266,10.148,149.556
C01457=1123.023,271.124,-72.928,-178.269,10.145,149.556
C01458=1123.027,270.876,-72.899,-178.272,10.143,149.556
C01459=1123.031,270.627,-72.869,-178.275,10.140,149.556
C01460=1123.035,270.380,-72.839,-178.277,10.138,149.556
C01461=1123.039,270.131,-72.810,-178.280,10.135,149.556
C01462=1123.043,269.883,-72.780,-178.283,10.132,149.557
C01463=1123.047,269.635,-72.751,-178.286,10.130,149.557
C01464=1123.052,269.387,-72.721,-178.288,10.128,149.557
C01465=1123.056,269.138,-72.692,-178.291,10.125,149.557
C01466=1123.060,268.890,-72.662,-178.294,10.122,149.557
C01467=1123.065,268.642,-72.632,-178.297,10.119,149.557
C01468=1123.069,268.393,-72.603,-178.299,10.117,149.557
C01469=1123.073,268.145,-72.573,-178.302,10.115,149.557
C01470=1123.077,267.897,-72.544,-178.305,10.113,149.557
C01471=1123.081,267.683,-72.519,-178.308,10.110,149.558
C01472=1123.084,267.471,-72.493,-178.309,10.107,149.558
C01473=1123.088,267.257,-72.468,-178.312,10.105,149.558
C01474=1123.091,267.044,-72.443,-178.314,10.104,149.558
C01475=1123.095,266.830,-72.417,-178.316,10.102,149.558
C01476=1123.099,266.617,-72.392,-178.319,10.100,149.558
C01477=1123.103,266.404,-72.367,-178.321,10.097,149.558
C01478=1123.106,266.191,-72.342,-178.323,10.095,149.558
C01479=1123.110,265.942,-72.313,-178.326,10.092,149.558
C01480=1123.115,265.694,-72.283,-178.328,10.090,149.558
C01481=1123.119,265.446,-72.254,-178.331,10.088,149.558
C01482=1123.123,265.198,-72.224,-178.333,10.086,149.559
C01483=1123.127,264.949,-72.196,-178.336,10.083,149.559
C01484=1123.132,264.700,-72.166,-178.339,10.081,149.559
C01485=1123.136,264.452,-72.137,-178.342,10.078,149.559
C01486=1123.141,264.205,-72.108,-178.345,10.075,149.559
C01487=1123.145,263.956,-72.078,-178.349,10.072,149.559
C01488=1123.149,263.708,-72.049,-178.352,10.070,149.560
C01489=1123.153,263.459,-72.020,-178.355,10.066,149.560
C01490=1123.157,263.211,-71.991,-178.359,10.063,149.560
C01491=1123.161,262.963,-71.962,-178.362,10.060,149.560
C01492=1123.166,262.715,-71.933,-178.366,10.057,149.560
C01493=1123.170,262.467,-71.904,-178.369,10.055,149.560
C01494=1123.175,262.218,-71.874,-178.373,10.052,149.561
C01495=1123.179,261.970,-71.845,-178.376,10.049,149.561
C01496=1123.182,261.721,-71.817,-178.379,10.046,149.561
C01497=1123.187,261.474,-71.788,-178.383,10.043,149.561
C01498=1123.191,261.226,-71.758,-178.386,10.040,149.561
C01499=1123.196,260.977,-71.730,-178.390,10.036,149.561
C01500=1123.200,260.728,-71.700,-178.393,10.034,149.562
C01501=1123.204,260.480,-71.672,-178.396,10.031,149.562
C01502=1123.209,260.232,-71.643,-178.400,10.028,149.562
C01503=1123.213,259.984,-71.613,-178.402,10.025,149.562
C01504=1123.217,259.735,-71.585,-178.405,10.022,149.562
C01505=1123.221,259.487,-71.556,-178.408,10.019,149.562
C01506=1123.226,259.239,-71.527,-178.412,10.016,149.562
C01507=1123.230,258.991,-71.498,-178.415,10.013,149.562
C01508=1123.234,258.742,-71.470,-178.418,10.010,149.563
C01509=1123.238,258.494,-71.440,-178.421,10.008,149.563
C01510=1123.243,258.246,-71.412,-178.424,10.005,149.563
C01511=1123.246,257.998,-71.383,-178.427,10.002,149.563
C01512=1123.251,257.749,-71.354,-178.430,9.999,149.563
C01513=1123.256,257.501,-71.326,-178.433,9.996,149.563
C01514=1123.259,257.253,-71.297,-178.436,9.993,149.563
C01515=1123.264,257.004,-71.268,-178.439,9.990,149.563
C01516=1123.269,256.756,-71.239,-178.442,9.987,149.563
C01517=1123.273,256.508,-71.211,-178.445,9.984,149.563
C01518=1123.277,256.259,-71.183,-178.447,9.982,149.563
C01519=1123.281,256.012,-71.154,-178.450,9.979,149.564
C01520=1123.286,255.763,-71.125,-178.451,9.978,149.563
C01521=1123.290,255.514,-71.097,-178.451,9.977,149.563
C01522=1123.294,255.267,-71.068,-178.451,9.976,149.563
C01523=1123.299,255.018,-71.039,-178.452,9.974,149.563
C01524=1123.302,254.769,-71.011,-178.453,9.973,149.563
C01525=1123.307,254.521,-70.982,-178.453,9.971,149.562
C01526=1123.311,254.273,-70.954,-178.455,9.969,149.562
C01527=1123.315,254.059,-70.929,-178.456,9.968,149.562
C01528=1123.318,253.845,-70.904,-178.458,9.967,149.562
C01529=1123.323,253.632,-70.880,-178.459,9.965,149.562
C01530=1123.326,253.419,-70.856,-178.461,9.963,149.562
C01531=1123.329,253.205,-70.831,-178.462,9.961,149.562
C01532=1123.334,252.992,-70.806,-178.464,9.959,149.562
C01533=1123.337,252.779,-70.782,-178.466,9.958,149.563
C01534=1123.340,252.565,-70.757,-178.468,9.956,149.563
C01535=1123.345,252.317,-70.729,-178.471,9.953,149.563
C01536=1123.349,252.068,-70.701,-178.474,9.951,149.563
C01537=1123.354,251.819,-70.672,-178.477,9.949,149.563
C01538=1123.358,251.572,-70.644,-178.480,9.945,149.563
C01539=1123.362,251.323,-70.615,-178.484,9.943,149.564
C01540=1123.367,251.075,-70.587,-178.487,9.941,149.564
C01541=1123.371,250.827,-70.558,-178.491,9.937,149.564
C01542=1123.375,250.578,-70.530,-178.495,9.934,149.565
C01543=1123.379,250.330,-70.502,-178.499,9.931,149.565
C01544=1123.384,250.081,-70.474,-178.504,9.927,149.565
C01545=1123.388,249.833,-70.446,-178.508,9.924,149.565
C01546=1123.392,249.584,-70.417,-178.513,9.920,149.566
C01547=1123.397,249.337,-70.389,-178.517,9.916,149.566
C01548=1123.401,249.088,-70.361,-178.522,9.912,149.566
C01549=1123.405,248.839,-70.332,-178.528,9.908,149.567
C01550=1123.409,248.591,-70.305,-178.533,9.904,149.567
C01551=1123.413,248.343,-70.277,-178.538,9.900,149.568
C01552=1123.418,248.094,-70.248,-178.544,9.895,149.568
C01553=1123.422,247.846,-70.220,-178.550,9.890,149.568
C01554=1123.426,247.598,-70.192,-178.556,9.885,149.569
C01555=1123.431,247.350,-70.164,-178.560,9.882,149.569
C01556=1123.435,247.101,-70.136,-178.562,9.879,149.569
C01557=1123.440,246.853,-70.109,-178.563,9.877,149.569
C01558=1123.444,246.604,-70.081,-178.565,9.875,149.569
C01559=1123.449,246.356,-70.052,-178.566,9.873,149.569
C01560=1123.452,246.107,-70.024,-178.568,9.870,149.568
C01561=1123.457,245.859,-69.997,-178.570,9.868,149.568
C01562=1123.461,245.610,-69.969,-178.572,9.865,149.568
C01563=1123.466,245.362,-69.940,-178.574,9.863,149.568
C01564=1123.470,245.114,-69.913,-178.574,9.861,149.568
C01565=1123.474,244.865,-69.885,-178.576,9.859,149.568
C01566=1123.479,244.617,-69.857,-178.578,9.856,149.568
C01567=1123.482,244.369,-69.829,-178.580,9.854,149.568
C01568=1123.487,244.120,-69.801,-178.582,9.852,149.568
C01569=1123.492,243.871,-69.773,-178.584,9.849,149.568
C01570=1123.496,243.623,-69.746,-178.586,9.847,149.568
C01571=1123.500,243.375,-69.718,-178.588,9.845,149.568
C01572=1123.504,243.126,-69.691,-178.590,9.843,149.568
C01573=1123.509,242.878,-69.663,-178.593,9.840,149.568
C01574=1123.513,242.630,-69.634,-178.594,9.837,149.568
C01575=1123.518,242.381,-69.607,-178.596,9.835,149.567
C01576=1123.522,242.133,-69.579,-178.599,9.833,149.568
C01577=1123.526,241.885,-69.551,-178.601,9.831,149.568
C01578=1123.531,241.636,-69.524,-178.603,9.828,149.567
C01579=1123.534,241.387,-69.496,-178.605,9.826,149.568
C01580=1123.539,241.139,-69.469,-178.607,9.823,149.568
C01581=1123.543,240.891,-69.441,-178.610,9.821,149.568
C01582=1123.547,240.642,-69.414,-178.612,9.818,149.568
C01583=1123.552,240.429,-69.389,-178.614,9.816,149.568
C01584=1123.555,240.215,-69.366,-178.616,9.814,149.568
C01585=1123.559,240.002,-69.342,-178.618,9.813,149.568
C01586=1123.563,239.788,-69.318,-178.620,9.810,149.568
C01587=1123.567,239.574,-69.295,-178.622,9.808,149.568
C01588=1123.570,239.360,-69.271,-178.624,9.806,149.568
C01589=1123.574,239.147,-69.247,-178.626,9.804,149.568
C01590=1123.578,238.934,-69.223,-178.628,9.802,149.568
C01591=1123.582,238.685,-69.196,-178.631,9.799,149.568
C01592=1123.586,238.437,-69.168,-178.634,9.796,149.568
C01593=1123.591,238.188,-69.141,-178.636,9.794,149.568
C01594=1123.595,237.940,-69.113,-178.639,9.791,149.568
C01595=1123.599,237.691,-69.086,-178.641,9.789,149.568
C01596=1123.604,237.443,-69.059,-178.644,9.786,149.569
C01597=1123.608,237.194,-69.031,-178.647,9.783,149.568
C01598=1123.612,236.946,-69.004,-178.650,9.781,149.569
C01599=1123.617,236.698,-68.976,-178.652,9.779,149.569
C01600=1123.621,236.449,-68.949,-178.655,9.776,149.569
C01601=1123.626,236.200,-68.921,-178.658,9.773,149.569
C01602=1123.630,235.952,-68.894,-178.661,9.770,149.569
C01603=1123.635,235.704,-68.867,-178.664,9.768,149.569
C01604=1123.639,235.455,-68.839,-178.667,9.765,149.569
C01605=1123.643,235.207,-68.813,-178.669,9.762,149.569
C01606=1123.647,234.959,-68.785,-178.672,9.759,149.569
C01607=1123.652,234.710,-68.758,-178.675,9.756,149.570
C01608=1123.656,234.462,-68.731,-178.678,9.753,149.570
C01609=1123.660,234.212,-68.703,-178.681,9.751,149.570
C01610=1123.665,233.965,-68.676,-178.684,9.748,149.570
C01611=1123.669,233.716,-68.648,-178.687,9.745,149.570
C01612=1123.674,233.468,-68.621,-178.690,9.743,149.570
C01613=1123.677,233.219,-68.595,-178.694,9.739,149.570
C01614=1123.682,232.970,-68.567,-178.697,9.736,149.570
C01615=1123.687,232.722,-68.540,-178.699,9.733,149.571
C01616=1123.691,232.474,-68.513,-178.702,9.731,149.571
C01617=1123.696,232.225,-68.486,-178.706,9.727,149.571
C01618=1123.699,231.977,-68.459,-178.709,9.724,149.571
C01619=1123.704,231.728,-68.432,-178.713,9.721,149.571
C01620=1123.708,231.479,-68.405,-178.715,9.718,149.571
C01621=1123.713,231.231,-68.378,-178.719,9.715,149.571
C01622=1123.717,230.982,-68.351,-178.722,9.712,149.572
C01623=1123.721,230.734,-68.324,-178.726,9.709,149.572
C01624=1123.726,230.486,-68.297,-178.729,9.706,149.572
C01625=1123.731,230.237,-68.270,-178.733,9.702,149.572
C01626=1123.734,229.988,-68.243,-178.736,9.699,149.572
C01627=1123.739,229.740,-68.216,-178.740,9.695,149.572
C01628=1123.743,229.491,-68.189,-178.743,9.693,149.572
C01629=1123.748,229.243,-68.162,-178.746,9.689,149.572
C01630=1123.752,228.995,-68.135,-178.750,9.686,149.573
C01631=1123.757,228.746,-68.108,-178.753,9.683,149.573
C01632=1123.761,228.498,-68.081,-178.756,9.679,149.573
C01633=1123.765,228.249,-68.056,-178.759,9.676,149.573
C01634=1123.770,228.000,-68.029,-178.762,9.673,149.573
C01635=1123.774,227.752,-68.002,-178.766,9.669,149.573
C01636=1123.779,227.504,-67.975,-178.770,9.666,149.573
C01637=1123.783,227.255,-67.948,-178.772,9.663,149.573
C01638=1123.787,227.006,-67.922,-178.776,9.659,149.573
C01639=1123.791,226.793,-67.898,-178.779,9.656,149.573
C01640=1123.795,226.579,-67.876,-178.781,9.653,149.573
C01641=1123.799,226.365,-67.853,-178.784,9.651,149.573
C01642=1123.802,226.151,-67.830,-178.786,9.648,149.573
C01643=1123.806,225.937,-67.807,-178.789,9.645,149.573
C01644=1123.810,225.724,-67.785,-178.792,9.642,149.573
C01645=1123.814,225.510,-67.762,-178.794,9.639,149.573
C01646=1123.818,225.297,-67.739,-178.797,9.636,149.573
C01647=1123.822,225.048,-67.712,-178.800,9.633,149.573
C01648=1123.826,224.800,-67.685,-178.802,9.630,149.573
C01649=1123.831,224.551,-67.659,-178.806,9.627,149.573
C01650=1123.835,224.303,-67.633,-178.808,9.624,149.573
C01651=1123.840,224.054,-67.606,-178.811,9.620,149.573
C01652=1123.844,223.806,-67.580,-178.814,9.617,149.573
C01653=1123.849,223.557,-67.553,-178.817,9.614,149.573
C01654=1123.853,223.308,-67.527,-178.819,9.611,149.573
C01655=1123.857,223.060,-67.501,-178.822,9.607,149.573
C01656=1123.862,222.811,-67.474,-178.825,9.604,149.573
C01657=1123.866,222.563,-67.448,-178.828,9.601,149.573
C01658=1123.871,222.314,-67.421,-178.830,9.598,149.573
C01659=1123.875,222.065,-67.395,-178.833,9.595,149.573
C01660=1123.880,221.816,-67.369,-178.836,9.592,149.573
C01661=1123.883,221.568,-67.342,-178.838,9.589,149.573
C01662=1123.888,221.319,-67.316,-178.841,9.585,149.573
C01663=1123.892,221.071,-67.289,-178.844,9.582,149.573
C01664=1123.897,220.823,-67.264,-178.846,9.578,149.573
C01665=1123.901,220.574,-67.238,-178.849,9.575,149.573
C01666=1123.906,220.325,-67.211,-178.851,9.572,149.572
C01667=1123.910,220.077,-67.185,-178.853,9.569,149.572
C01668=1123.914,219.828,-67.159,-178.856,9.566,149.572
C01669=1123.919,219.579,-67.133,-178.858,9.563,149.572
C01670=1123.923,219.331,-67.107,-178.860,9.560,149.572
C01671=1123.927,219.082,-67.080,-178.863,9.557,149.572
C01672=1123.933,218.834,-67.054,-178.865,9.554,149.572
C01673=1123.937,218.585,-67.029,-178.868,9.551,149.572
C01674=1123.941,218.337,-67.002,-178.870,9.547,149.572
C01675=1123.945,218.088,-66.976,-178.873,9.544,149.572
C01676=1123.950,217.839,-66.950,-178.874,9.542,149.572
C01677=1123.954,217.590,-66.924,-178.877,9.539,149.571
C01678=1123.958,217.342,-66.898,-178.879,9.535,149.571
C01679=1123.963,217.094,-66.872,-178.881,9.533,149.571
C01680=1123.967,216.845,-66.847,-178.883,9.530,149.571
C01681=1123.972,216.596,-66.820,-178.886,9.527,149.571
C01682=1123.977,216.347,-66.795,-178.888,9.524,149.571
C01683=1123.980,216.099,-66.768,-178.890,9.521,149.571
C01684=1123.985,215.851,-66.743,-178.892,9.518,149.571
C01685=1123.990,215.602,-66.717,-178.894,9.515,149.571
C01686=1123.994,215.353,-66.691,-178.896,9.513,149.570
C01687=1123.999,215.104,-66.665,-178.898,9.509,149.570
C01688=1124.003,214.855,-66.639,-178.900,9.507,149.570
C01689=1124.007,214.608,-66.613,-178.902,9.504,149.570
C01690=1124.012,214.359,-66.587,-178.904,9.501,149.570
C01691=1124.016,214.110,-66.562,-178.905,9.499,149.570
C01692=1124.021,213.861,-66.535,-178.908,9.496,149.570
C01693=1124.026,213.613,-66.510,-178.909,9.493,149.569
C01694=1124.030,213.364,-66.484,-178.911,9.490,149.569
C01695=1124.033,213.151,-66.462,-178.913,9.488,149.569
C01696=1124.038,212.937,-66.440,-178.915,9.485,149.569
C01697=1124.041,212.723,-66.418,-178.917,9.483,149.569
C01698=1124.045,212.509,-66.396,-178.918,9.481,149.569
C01699=1124.049,212.296,-66.373,-178.920,9.478,149.569
C01700=1124.053,212.081,-66.351,-178.922,9.476,149.569
C01701=1124.056,211.867,-66.330,-178.924,9.474,149.569
C01702=1124.061,211.654,-66.307,-178.926,9.471,149.568
C01703=1124.065,211.405,-66.281,-178.928,9.469,149.568
C01704=1124.069,211.156,-66.255,-178.930,9.466,149.568
C01705=1124.073,210.907,-66.230,-178.932,9.463,149.568
C01706=1124.078,210.659,-66.204,-178.935,9.461,149.568
C01707=1124.082,210.411,-66.179,-178.937,9.458,149.568
C01708=1124.086,210.162,-66.153,-178.939,9.455,149.568
C01709=1124.091,209.914,-66.127,-178.941,9.453,149.568
C01710=1124.096,209.664,-66.102,-178.944,9.450,149.568
C01711=1124.100,209.415,-66.077,-178.946,9.447,149.568
C01712=1124.105,209.167,-66.051,-178.949,9.445,149.568
C01713=1124.109,208.918,-66.026,-178.951,9.442,149.568
C01714=1124.113,208.670,-66.000,-178.954,9.438,149.568
C01715=1124.118,208.422,-65.974,-178.956,9.436,149.568
C01716=1124.122,208.173,-65.949,-178.958,9.433,149.568
C01717=1124.127,207.923,-65.924,-178.961,9.431,149.569
C01718=1124.132,207.675,-65.898,-178.964,9.427,149.568
C01719=1124.136,207.426,-65.872,-178.966,9.426,149.569
C01720=1124.140,207.178,-65.847,-178.969,9.422,149.569
C01721=1124.145,206.930,-65.821,-178.972,9.420,149.569
C01722=1124.150,206.680,-65.796,-178.974,9.417,149.569
C01723=1124.154,206.432,-65.771,-178.977,9.414,149.569
C01724=1124.159,206.183,-65.745,-178.980,9.411,149.569
C01725=1124.162,205.934,-65.721,-178.983,9.408,149.569
C01726=1124.167,205.686,-65.695,-178.986,9.405,149.569
C01727=1124.171,205.437,-65.670,-178.989,9.402,149.569
C01728=1124.176,205.189,-65.644,-178.991,9.399,149.569
C01729=1124.181,204.940,-65.619,-178.994,9.397,149.569
C01730=1124.185,204.691,-65.593,-178.997,9.394,149.569
C01731=1124.190,204.442,-65.569,-179.000,9.391,149.570
C01732=1124.194,204.194,-65.544,-179.003,9.388,149.570
C01733=1124.198,203.946,-65.518,-179.005,9.385,149.570
C01734=1124.203,203.696,-65.493,-179.008,9.383,149.570
C01735=1124.208,203.448,-65.468,-179.012,9.379,149.570
C01736=1124.212,203.199,-65.443,-179.015,9.376,149.570
C01737=1124.217,202.950,-65.417,-179.018,9.374,149.570
C01738=1124.221,202.701,-65.393,-179.021,9.370,149.570
C01739=1124.226,202.453,-65.368,-179.024,9.367,149.570
C01740=1124.230,202.204,-65.343,-179.027,9.364,149.570
C01741=1124.234,201.955,-65.317,-179.031,9.361,149.571
C01742=1124.239,201.707,-65.293,-179.033,9.358,149.571
C01743=1124.243,201.458,-65.267,-179.037,9.354,149.571
C01744=1124.248,201.209,-65.242,-179.040,9.352,149.571
C01745=1124.252,200.961,-65.217,-179.044,9.348,149.571
C01746=1124.257,200.712,-65.192,-179.047,9.345,149.571
C01747=1124.261,200.463,-65.167,-179.050,9.342,149.571
C01748=1124.266,200.215,-65.143,-179.053,9.339,149.571
C01749=1124.271,199.966,-65.118,-179.056,9.335,149.572
C01750=1124.275,199.717,-65.092,-179.060,9.332,149.572
C01751=1124.278,199.503,-65.071,-179.063,9.329,149.572
C01752=1124.282,199.289,-65.050,-179.066,9.326,149.572
C01753=1124.287,199.075,-65.029,-179.069,9.324,149.572
C01754=1124.290,198.861,-65.007,-179.071,9.320,149.572
C01755=1124.294,198.647,-64.986,-179.074,9.318,149.572
C01756=1124.297,198.433,-64.964,-179.077,9.315,149.572
C01757=1124.302,198.220,-64.944,-179.081,9.311,149.573
C01758=1124.306,198.006,-64.923,-179.083,9.308,149.572
C01759=1124.310,197.756,-64.897,-179.087,9.305,149.573
C01760=1124.315,197.508,-64.872,-179.090,9.301,149.573
C01761=1124.319,197.260,-64.848,-179.094,9.298,149.573
C01762=1124.324,197.010,-64.823,-179.098,9.294,149.573
C01763=1124.328,196.762,-64.799,-179.101,9.290,149.573
C01764=1124.333,196.512,-64.774,-179.104,9.287,149.573
C01765=1124.337,196.264,-64.750,-179.108,9.283,149.573
C01766=1124.342,196.015,-64.725,-179.109,9.281,149.573
C01767=1124.346,195.767,-64.700,-179.111,9.278,149.573
C01768=1124.351,195.518,-64.675,-179.113,9.276,149.573
C01769=1124.355,195.270,-64.651,-179.114,9.273,149.572
C01770=1124.360,195.020,-64.626,-179.116,9.271,149.572
C01771=1124.364,194.772,-64.602,-179.118,9.268,149.572
C01772=1124.369,194.523,-64.578,-179.119,9.266,149.572
C01773=1124.373,194.274,-64.553,-179.122,9.262,149.572
C01774=1124.378,194.026,-64.529,-179.123,9.260,149.572
C01775=1124.383,193.777,-64.504,-179.125,9.257,149.572
C01776=1124.386,193.528,-64.480,-179.127,9.255,149.572
C01777=1124.392,193.279,-64.455,-179.128,9.252,149.571
C01778=1124.396,193.031,-64.431,-179.130,9.250,149.571
C01779=1124.400,192.782,-64.407,-179.133,9.247,149.571
C01780=1124.405,192.533,-64.382,-179.134,9.244,149.571
C01781=1124.409,192.284,-64.358,-179.136,9.242,149.571
C01782=1124.414,192.036,-64.333,-179.139,9.238,149.571
C01783=1124.418,191.786,-64.309,-179.140,9.236,149.571
C01784=1124.423,191.538,-64.285,-179.142,9.233,149.571
C01785=1124.428,191.289,-64.260,-179.144,9.230,149.571
